LIN {X 0.189,Y -441.248,Z 653.481,A 0.000,B 0.000,C 90.000,E1 266.560} C_DIS
LIN {X -0.054,Y -433.305,Z 653.480,A 0.000,B 0.000,C 90.000,E1 266.388} C_DIS
LIN {X 0.144,Y -424.174,Z 653.479,A 0.000,B 0.000,C 90.000,E1 266.216} C_DIS
LIN {X 0.128,Y -416.575,Z 653.479,A 0.000,B 0.000,C 90.000,E1 266.159} C_DIS
LIN {X 0.071,Y -413.712,Z 653.479,A 0.000,B 0.000,C 90.000,E1 266.159} C_DIS
LIN {X 0.007,Y -180.928,Z 653.479,A 0.000,B 0.000,C 90.000,E1 266.159} C_DIS
LIN {X -0.082,Y -180.902,Z 653.474,A 0.000,B 0.000,C 90.000,E1 265.298} C_DIS
LIN {X 0.047,Y -180.232,Z 653.464,A 0.000,B 0.000,C 90.000,E1 263.571} C_DIS
LIN {X 0.064,Y -178.714,Z 653.441,A 0.000,B 0.000,C 90.000,E1 259.342} C_DIS
LIN {X -0.044,Y -175.764,Z 653.413,A 0.000,B 0.000,C 90.000,E1 254.283} C_DIS
LIN {X 0.006,Y -171.947,Z 653.384,A 0.000,B 0.000,C 90.000,E1 249.135} C_DIS
LIN {X -0.018,Y -171.334,Z 653.379,A 0.000,B 0.000,C 90.000,E1 248.284} C_DIS
LIN {X 0.034,Y -167.588,Z 653.355,A 0.000,B 0.000,C 90.000,E1 243.948} C_DIS
LIN {X -0.026,Y -166.226,Z 653.346,A 0.000,B 0.000,C 90.000,E1 242.231} C_DIS
LIN {X -0.038,Y -162.987,Z 653.326,A 0.000,B 0.000,C 90.000,E1 238.742} C_DIS
LIN {X 0.009,Y -160.904,Z 653.312,A 0.000,B 0.000,C 90.000,E1 236.087} C_DIS
LIN {X -0.013,Y -157.670,Z 653.292,A 0.000,B 0.000,C 90.000,E1 232.557} C_DIS
LIN {X -0.075,Y -155.708,Z 653.277,A 0.000,B 0.000,C 90.000,E1 229.908} C_DIS
LIN {X -0.020,Y -151.971,Z 653.252,A 0.000,B 0.000,C 90.000,E1 225.405} C_DIS
LIN {X -0.004,Y -150.213,Z 653.237,A 0.000,B 0.000,C 90.000,E1 222.690} C_DIS
LIN {X -0.079,Y -146.978,Z 653.212,A 0.000,B 0.000,C 90.000,E1 218.177} C_DIS
LIN {X 0.030,Y -145.565,Z 653.197,A 0.000,B 0.000,C 90.000,E1 215.391} C_DIS
LIN {X 0.029,Y -142.956,Z 653.171,A 0.000,B 0.000,C 90.000,E1 210.797} C_DIS
LIN {X -0.041,Y -141.582,Z 653.151,A 0.000,B 0.000,C 90.000,E1 207.129} C_DIS
LIN {X 0.007,Y -139.416,Z 653.115,A 0.000,B 0.000,C 90.000,E1 200.610} C_DIS
LIN {X 0.059,Y -139.142,Z 653.104,A 0.000,B 0.000,C 90.000,E1 198.725} C_DIS
LIN {X -0.050,Y -138.348,Z 653.057,A 0.000,B 0.000,C 90.000,E1 190.366} C_DIS
LIN {X -0.065,Y -139.491,Z 653.006,A 0.000,B 0.000,C 90.000,E1 181.031} C_DIS
LIN {X 0.015,Y -141.101,Z 652.975,A 0.000,B 0.000,C 90.000,E1 175.412} C_DIS
LIN {X -0.031,Y -142.479,Z 652.959,A 0.000,B 0.000,C 90.000,E1 172.648} C_DIS
LIN {X 0.058,Y -144.728,Z 652.933,A 0.000,B 0.000,C 90.000,E1 167.993} C_DIS
LIN {X 0.009,Y -147.332,Z 652.913,A 0.000,B 0.000,C 90.000,E1 164.338} C_DIS
LIN {X 0.074,Y -150.655,Z 652.888,A 0.000,B 0.000,C 90.000,E1 159.752} C_DIS
LIN {X -0.045,Y -154.133,Z 652.868,A 0.000,B 0.000,C 90.000,E1 156.177} C_DIS
LIN {X 0.018,Y -157.560,Z 652.848,A 0.000,B 0.000,C 90.000,E1 152.564} C_DIS
LIN {X 0.042,Y -161.803,Z 652.828,A 0.000,B 0.000,C 90.000,E1 148.997} C_DIS
LIN {X 0.062,Y -165.995,Z 652.808,A 0.000,B 0.000,C 90.000,E1 145.468} C_DIS
LIN {X 0.055,Y -170.992,Z 652.789,A 0.000,B 0.000,C 90.000,E1 141.984} C_DIS
LIN {X -0.029,Y -175.862,Z 652.770,A 0.000,B 0.000,C 90.000,E1 138.566} C_DIS
LIN {X -0.035,Y -181.467,Z 652.751,A 0.000,B 0.000,C 90.000,E1 135.162} C_DIS
LIN {X 0.101,Y -186.979,Z 652.732,A 0.000,B 0.000,C 90.000,E1 131.757} C_DIS
LIN {X -0.120,Y -191.043,Z 652.720,A 0.000,B 0.000,C 90.000,E1 129.644} C_DIS
LIN {X 0.173,Y -288.470,Z 652.720,A 0.000,B 0.000,C 90.000,E1 129.564} C_DIS
LIN {X 0.015,Y -290.425,Z 652.720,A 0.000,B 0.000,C 90.000,E1 129.564} C_DIS
LIN {X 0.087,Y -295.635,Z 652.718,A 0.000,B 0.000,C 90.000,E1 129.277} C_DIS
LIN {X -0.103,Y -298.817,Z 652.716,A 0.000,B 0.000,C 90.000,E1 128.991} C_DIS
LIN {X 0.074,Y -302.429,Z 652.713,A 0.000,B 0.000,C 90.000,E1 128.382} C_DIS
LIN {X -0.165,Y -303.887,Z 652.711,A 0.000,B 0.000,C 90.000,E1 128.096} C_DIS
LIN {X 0.022,Y -305.034,Z 652.710,A 0.000,B 0.000,C 90.000,E1 127.729} C_DIS
LIN {X 0.132,Y -315.593,Z 652.690,A 0.000,B 0.000,C 90.000,E1 124.119} C_DIS
LIN {X 0.009,Y -325.562,Z 652.674,A 0.000,B 0.000,C 90.000,E1 121.258} C_DIS
LIN {X -0.046,Y -336.851,Z 652.658,A 0.000,B 0.000,C 90.000,E1 118.437} C_DIS
LIN {X -0.093,Y -349.566,Z 652.643,A 0.000,B 0.000,C 90.000,E1 115.668} C_DIS
LIN {X -0.148,Y -362.154,Z 652.629,A 0.000,B 0.000,C 90.000,E1 113.259} C_DIS
LIN {X 0.024,Y -376.047,Z 652.616,A 0.000,B 0.000,C 90.000,E1 110.865} C_DIS
LIN {X 0.075,Y -391.345,Z 652.603,A 0.000,B 0.000,C 90.000,E1 108.544} C_DIS
LIN {X -0.132,Y -408.159,Z 652.591,A 0.000,B 0.000,C 90.000,E1 106.315} C_DIS
LIN {X -0.168,Y -426.613,Z 652.578,A 0.000,B 0.000,C 90.000,E1 104.120} C_DIS
LIN {X -0.103,Y -446.484,Z 652.567,A 0.000,B 0.000,C 90.000,E1 102.007} C_DIS
LIN {X -0.102,Y -466.963,Z 652.556,A 0.000,B 0.000,C 90.000,E1 100.074} C_DIS
LIN {X -0.128,Y -469.546,Z 652.555,A 0.000,B 0.000,C 90.000,E1 99.849} C_DIS
LIN {X -0.072,Y -471.802,Z 652.553,A 0.000,B 0.000,C 90.000,E1 99.613} C_DIS
LIN {X -0.186,Y -473.637,Z 652.552,A 0.000,B 0.000,C 90.000,E1 99.378} C_DIS
LIN {X 0.092,Y -475.022,Z 652.551,A 0.000,B 0.000,C 90.000,E1 99.095} C_DIS
LIN {X -0.185,Y -476.807,Z 652.548,A 0.000,B 0.000,C 90.000,E1 98.624} C_DIS
LIN {X -0.055,Y -477.505,Z 652.545,A 0.000,B 0.000,C 90.000,E1 98.106} C_DIS
LIN {X 0.087,Y -477.233,Z 652.542,A 0.000,B 0.000,C 90.000,E1 97.587} C_DIS
LIN {X -0.237,Y -475.951,Z 652.539,A 0.000,B 0.000,C 90.000,E1 97.125} C_DIS
LIN {X 0.100,Y -474.870,Z 652.538,A 0.000,B 0.000,C 90.000,E1 96.834} C_DIS
LIN {X -0.091,Y -473.421,Z 652.537,A 0.000,B 0.000,C 90.000,E1 96.606} C_DIS
LIN {X -0.133,Y -456.317,Z 652.523,A 0.000,B 0.000,C 90.000,E1 94.073} C_DIS
LIN {X 0.065,Y -445.602,Z 652.512,A 0.000,B 0.000,C 90.000,E1 92.236} C_DIS
LIN {X 0.026,Y -435.545,Z 652.502,A 0.000,B 0.000,C 90.000,E1 90.401} C_DIS
LIN {X 0.069,Y -426.626,Z 652.493,A 0.000,B 0.000,C 90.000,E1 88.797} C_DIS
LIN {X 0.061,Y -415.774,Z 652.483,A 0.000,B 0.000,C 90.000,E1 86.906} C_DIS
LIN {X 0.035,Y -401.764,Z 652.469,A 0.000,B 0.000,C 90.000,E1 84.432} C_DIS
LIN {X 0.082,Y -388.231,Z 652.455,A 0.000,B 0.000,C 90.000,E1 81.894} C_DIS
LIN {X -0.121,Y -375.167,Z 652.441,A 0.000,B 0.000,C 90.000,E1 79.342} C_DIS
LIN {X -0.091,Y -362.604,Z 652.426,A 0.000,B 0.000,C 90.000,E1 76.700} C_DIS
LIN {X 0.082,Y -348.061,Z 652.408,A 0.000,B 0.000,C 90.000,E1 73.378} C_DIS
LIN {X 0.057,Y -334.377,Z 652.389,A 0.000,B 0.000,C 90.000,E1 70.007} C_DIS
LIN {X 0.031,Y -321.830,Z 652.370,A 0.000,B 0.000,C 90.000,E1 66.561} C_DIS
LIN {X -0.103,Y -309.547,Z 652.348,A 0.000,B 0.000,C 90.000,E1 62.743} C_DIS
LIN {X 0.008,Y -300.306,Z 652.330,A 0.000,B 0.000,C 90.000,E1 59.459} C_DIS
LIN {X 0.042,Y -291.828,Z 652.312,A 0.000,B 0.000,C 90.000,E1 56.135} C_DIS
LIN {X 0.058,Y -283.710,Z 652.293,A 0.000,B 0.000,C 90.000,E1 52.763} C_DIS
LIN {X 0.008,Y -280.513,Z 652.286,A 0.000,B 0.000,C 90.000,E1 51.412} C_DIS
LIN {X -0.126,Y -277.134,Z 652.278,A 0.000,B 0.000,C 90.000,E1 50.070} C_DIS
LIN {X -0.128,Y -271.683,Z 652.267,A 0.000,B 0.000,C 90.000,E1 48.000} C_DIS
LIN {X -0.050,Y -265.784,Z 652.255,A 0.000,B 0.000,C 90.000,E1 45.891} C_DIS
LIN {X -0.089,Y -259.504,Z 652.243,A 0.000,B 0.000,C 90.000,E1 43.785} C_DIS
LIN {X 0.121,Y -252.929,Z 652.231,A 0.000,B 0.000,C 90.000,E1 41.595} C_DIS
LIN {X -0.104,Y -242.144,Z 652.211,A 0.000,B 0.000,C 90.000,E1 38.016} C_DIS
LIN {X 0.018,Y -234.162,Z 652.195,A 0.000,B 0.000,C 90.000,E1 35.025} C_DIS
LIN {X 0.056,Y -226.880,Z 652.178,A 0.000,B 0.000,C 90.000,E1 32.005} C_DIS
LIN {X 0.061,Y -220.310,Z 652.161,A 0.000,B 0.000,C 90.000,E1 28.949} C_DIS
LIN {X 0.078,Y -214.588,Z 652.144,A 0.000,B 0.000,C 90.000,E1 25.848} C_DIS
LIN {X 0.065,Y -209.634,Z 652.126,A 0.000,B 0.000,C 90.000,E1 22.717} C_DIS
LIN {X -0.026,Y -204.484,Z 652.104,A 0.000,B 0.000,C 90.000,E1 18.779} C_DIS
LIN {X -0.022,Y -200.459,Z 652.082,A 0.000,B 0.000,C 90.000,E1 14.773} C_DIS
LIN {X 0.038,Y -196.988,Z 652.055,A 0.000,B 0.000,C 90.000,E1 9.905} C_DIS
LIN {X 0.013,Y -194.464,Z 652.014,A 0.000,B 0.000,C 90.000,E1 2.579} C_DIS
LIN {X 0.002,Y -196.193,Z 651.961,A 0.000,B 0.000,C 90.000,E1 352.996} C_DIS
LIN {X 0.002,Y -199.224,Z 651.934,A 0.000,B 0.000,C 90.000,E1 348.117} C_DIS
LIN {X -0.079,Y -202.794,Z 651.912,A 0.000,B 0.000,C 90.000,E1 344.102} C_DIS
LIN {X 0.049,Y -207.381,Z 651.889,A 0.000,B 0.000,C 90.000,E1 340.061} C_DIS
LIN {X 0.033,Y -212.821,Z 651.867,A 0.000,B 0.000,C 90.000,E1 336.102} C_DIS
LIN {X -0.141,Y -218.987,Z 651.846,A 0.000,B 0.000,C 90.000,E1 332.231} C_DIS
LIN {X 0.089,Y -224.463,Z 651.828,A 0.000,B 0.000,C 90.000,E1 329.076} C_DIS
LIN {X 0.069,Y -231.711,Z 651.807,A 0.000,B 0.000,C 90.000,E1 325.261} C_DIS
LIN {X -0.086,Y -239.559,Z 651.786,A 0.000,B 0.000,C 90.000,E1 321.537} C_DIS
LIN {X 0.084,Y -248.181,Z 651.766,A 0.000,B 0.000,C 90.000,E1 317.796} C_DIS
LIN {X -0.049,Y -257.802,Z 651.745,A 0.000,B 0.000,C 90.000,E1 314.190} C_DIS
LIN {X -0.075,Y -267.404,Z 651.728,A 0.000,B 0.000,C 90.000,E1 310.987} C_DIS
LIN {X 0.177,Y -279.671,Z 651.708,A 0.000,B 0.000,C 90.000,E1 307.443} C_DIS
LIN {X -0.010,Y -293.237,Z 651.689,A 0.000,B 0.000,C 90.000,E1 304.072} C_DIS
LIN {X -0.002,Y -308.477,Z 651.671,A 0.000,B 0.000,C 90.000,E1 300.747} C_DIS
LIN {X -0.066,Y -323.517,Z 651.655,A 0.000,B 0.000,C 90.000,E1 297.847} C_DIS
LIN {X -0.144,Y -337.384,Z 651.641,A 0.000,B 0.000,C 90.000,E1 295.335} C_DIS
LIN {X 0.208,Y -355.656,Z 651.624,A 0.000,B 0.000,C 90.000,E1 292.206} C_DIS
LIN {X 0.158,Y -369.246,Z 651.612,A 0.000,B 0.000,C 90.000,E1 290.120} C_DIS
LIN {X -0.089,Y -384.236,Z 651.601,A 0.000,B 0.000,C 90.000,E1 288.109} C_DIS
LIN {X -0.200,Y -402.821,Z 651.588,A 0.000,B 0.000,C 90.000,E1 285.843} C_DIS
LIN {X -0.025,Y -414.425,Z 651.580,A 0.000,B 0.000,C 90.000,E1 284.426} C_DIS
LIN {X 0.081,Y -427.691,Z 651.571,A 0.000,B 0.000,C 90.000,E1 282.771} C_DIS
LIN {X 0.130,Y -438.189,Z 651.564,A 0.000,B 0.000,C 90.000,E1 281.422} C_DIS
LIN {X 0.108,Y -446.197,Z 651.558,A 0.000,B 0.000,C 90.000,E1 280.366} C_DIS
LIN {X 0.094,Y -454.150,Z 651.552,A 0.000,B 0.000,C 90.000,E1 279.321} C_DIS
LIN {X 0.057,Y -464.847,Z 651.545,A 0.000,B 0.000,C 90.000,E1 278.049} C_DIS
LIN {X -0.050,Y -470.598,Z 651.541,A 0.000,B 0.000,C 90.000,E1 277.296} C_DIS
LIN {X -0.104,Y -475.386,Z 651.536,A 0.000,B 0.000,C 90.000,E1 276.543} C_DIS
LIN {X -0.176,Y -479.394,Z 651.532,A 0.000,B 0.000,C 90.000,E1 275.796} C_DIS
LIN {X -0.027,Y -481.609,Z 651.529,A 0.000,B 0.000,C 90.000,E1 275.277} C_DIS
LIN {X 0.138,Y -483.468,Z 651.527,A 0.000,B 0.000,C 90.000,E1 274.759} C_DIS
LIN {X -0.213,Y -484.886,Z 651.524,A 0.000,B 0.000,C 90.000,E1 274.302} C_DIS
LIN {X -0.033,Y -485.902,Z 651.521,A 0.000,B 0.000,C 90.000,E1 273.784} C_DIS
LIN {X 0.125,Y -486.560,Z 651.518,A 0.000,B 0.000,C 90.000,E1 273.269} C_DIS
LIN {X -0.169,Y -486.874,Z 651.516,A 0.000,B 0.000,C 90.000,E1 272.808} C_DIS
LIN {X 0.002,Y -486.931,Z 651.513,A 0.000,B 0.000,C 90.000,E1 272.293} C_DIS
LIN {X 0.193,Y -486.719,Z 651.510,A 0.000,B 0.000,C 90.000,E1 271.776} C_DIS
LIN {X -0.120,Y -486.113,Z 651.507,A 0.000,B 0.000,C 90.000,E1 271.318} C_DIS
LIN {X 0.055,Y -485.118,Z 651.505,A 0.000,B 0.000,C 90.000,E1 270.802} C_DIS
LIN {X 0.226,Y -483.673,Z 651.502,A 0.000,B 0.000,C 90.000,E1 270.286} C_DIS
LIN {X -0.091,Y -481.651,Z 651.499,A 0.000,B 0.000,C 90.000,E1 269.828} C_DIS
LIN {X 0.066,Y -478.997,Z 651.496,A 0.000,B 0.000,C 90.000,E1 269.312} C_DIS
LIN {X 0.201,Y -475.487,Z 651.493,A 0.000,B 0.000,C 90.000,E1 268.797} C_DIS
LIN {X -0.156,Y -471.011,Z 651.491,A 0.000,B 0.000,C 90.000,E1 268.339} C_DIS
LIN {X 0.140,Y -468.359,Z 651.489,A 0.000,B 0.000,C 90.000,E1 268.051} C_DIS
LIN {X 0.024,Y -462.383,Z 651.487,A 0.000,B 0.000,C 90.000,E1 267.593} C_DIS
LIN {X 0.093,Y -459.096,Z 651.485,A 0.000,B 0.000,C 90.000,E1 267.364} C_DIS
LIN {X -0.043,Y -455.866,Z 651.484,A 0.000,B 0.000,C 90.000,E1 267.192} C_DIS
LIN {X 0.011,Y -448.763,Z 651.482,A 0.000,B 0.000,C 90.000,E1 266.846} C_DIS
LIN {X 0.165,Y -441.242,Z 651.481,A 0.000,B 0.000,C 90.000,E1 266.560} C_DIS
LIN {X -0.067,Y -433.363,Z 651.480,A 0.000,B 0.000,C 90.000,E1 266.388} C_DIS
LIN {X 0.125,Y -423.997,Z 651.479,A 0.000,B 0.000,C 90.000,E1 266.216} C_DIS
LIN {X 0.109,Y -415.978,Z 651.479,A 0.000,B 0.000,C 90.000,E1 266.159} C_DIS
LIN {X 0.052,Y -412.268,Z 651.479,A 0.000,B 0.000,C 90.000,E1 266.159} C_DIS
LIN {X -0.001,Y -180.927,Z 651.479,A 0.000,B 0.000,C 90.000,E1 266.159} C_DIS
LIN {X -0.088,Y -180.902,Z 651.474,A 0.000,B 0.000,C 90.000,E1 265.298} C_DIS
LIN {X 0.041,Y -180.231,Z 651.464,A 0.000,B 0.000,C 90.000,E1 263.571} C_DIS
LIN {X 0.058,Y -178.714,Z 651.441,A 0.000,B 0.000,C 90.000,E1 259.342} C_DIS
LIN {X -0.051,Y -175.762,Z 651.413,A 0.000,B 0.000,C 90.000,E1 254.283} C_DIS
LIN {X -0.001,Y -171.946,Z 651.384,A 0.000,B 0.000,C 90.000,E1 249.135} C_DIS
LIN {X -0.024,Y -171.332,Z 651.379,A 0.000,B 0.000,C 90.000,E1 248.284} C_DIS
LIN {X 0.029,Y -167.586,Z 651.355,A 0.000,B 0.000,C 90.000,E1 243.948} C_DIS
LIN {X -0.032,Y -166.224,Z 651.346,A 0.000,B 0.000,C 90.000,E1 242.231} C_DIS
LIN {X -0.044,Y -162.986,Z 651.326,A 0.000,B 0.000,C 90.000,E1 238.742} C_DIS
LIN {X 0.003,Y -160.901,Z 651.312,A 0.000,B 0.000,C 90.000,E1 236.087} C_DIS
LIN {X -0.018,Y -157.668,Z 651.292,A 0.000,B 0.000,C 90.000,E1 232.557} C_DIS
LIN {X -0.080,Y -155.706,Z 651.277,A 0.000,B 0.000,C 90.000,E1 229.908} C_DIS
LIN {X -0.026,Y -151.969,Z 651.252,A 0.000,B 0.000,C 90.000,E1 225.405} C_DIS
LIN {X -0.009,Y -150.211,Z 651.237,A 0.000,B 0.000,C 90.000,E1 222.690} C_DIS
LIN {X -0.085,Y -146.977,Z 651.212,A 0.000,B 0.000,C 90.000,E1 218.177} C_DIS
LIN {X 0.024,Y -145.563,Z 651.197,A 0.000,B 0.000,C 90.000,E1 215.391} C_DIS
LIN {X 0.023,Y -142.955,Z 651.171,A 0.000,B 0.000,C 90.000,E1 210.797} C_DIS
LIN {X -0.046,Y -141.581,Z 651.151,A 0.000,B 0.000,C 90.000,E1 207.129} C_DIS
LIN {X 0.002,Y -139.416,Z 651.115,A 0.000,B 0.000,C 90.000,E1 200.610} C_DIS
LIN {X 0.053,Y -139.141,Z 651.104,A 0.000,B 0.000,C 90.000,E1 198.725} C_DIS
LIN {X -0.055,Y -138.348,Z 651.057,A 0.000,B 0.000,C 90.000,E1 190.366} C_DIS
LIN {X 0.069,Y -139.491,Z 651.006,A 0.000,B 0.000,C 90.000,E1 180.974} C_DIS
LIN {X 0.010,Y -141.102,Z 650.975,A 0.000,B 0.000,C 90.000,E1 175.412} C_DIS
LIN {X -0.037,Y -142.480,Z 650.959,A 0.000,B 0.000,C 90.000,E1 172.648} C_DIS
LIN {X 0.052,Y -144.729,Z 650.933,A 0.000,B 0.000,C 90.000,E1 167.993} C_DIS
LIN {X 0.003,Y -147.334,Z 650.913,A 0.000,B 0.000,C 90.000,E1 164.338} C_DIS
LIN {X 0.068,Y -150.656,Z 650.888,A 0.000,B 0.000,C 90.000,E1 159.752} C_DIS
LIN {X -0.051,Y -154.135,Z 650.868,A 0.000,B 0.000,C 90.000,E1 156.177} C_DIS
LIN {X 0.012,Y -157.563,Z 650.848,A 0.000,B 0.000,C 90.000,E1 152.564} C_DIS
LIN {X 0.037,Y -161.806,Z 650.828,A 0.000,B 0.000,C 90.000,E1 148.997} C_DIS
LIN {X 0.056,Y -165.998,Z 650.808,A 0.000,B 0.000,C 90.000,E1 145.468} C_DIS
LIN {X 0.048,Y -170.995,Z 650.789,A 0.000,B 0.000,C 90.000,E1 141.984} C_DIS
LIN {X -0.036,Y -175.865,Z 650.770,A 0.000,B 0.000,C 90.000,E1 138.566} C_DIS
LIN {X -0.042,Y -181.470,Z 650.751,A 0.000,B 0.000,C 90.000,E1 135.162} C_DIS
LIN {X 0.094,Y -186.982,Z 650.732,A 0.000,B 0.000,C 90.000,E1 131.757} C_DIS
LIN {X -0.127,Y -191.046,Z 650.720,A 0.000,B 0.000,C 90.000,E1 129.644} C_DIS
LIN {X 0.162,Y -288.697,Z 650.720,A 0.000,B 0.000,C 90.000,E1 129.564} C_DIS
LIN {X 0.005,Y -290.478,Z 650.720,A 0.000,B 0.000,C 90.000,E1 129.564} C_DIS
LIN {X 0.077,Y -295.638,Z 650.718,A 0.000,B 0.000,C 90.000,E1 129.277} C_DIS
LIN {X 0.059,Y -298.836,Z 650.716,A 0.000,B 0.000,C 90.000,E1 128.955} C_DIS
LIN {X 0.038,Y -302.443,Z 650.713,A 0.000,B 0.000,C 90.000,E1 128.382} C_DIS
LIN {X 0.039,Y -303.894,Z 650.711,A 0.000,B 0.000,C 90.000,E1 128.051} C_DIS
LIN {X -0.014,Y -305.035,Z 650.710,A 0.000,B 0.000,C 90.000,E1 127.729} C_DIS
LIN {X 0.095,Y -315.593,Z 650.690,A 0.000,B 0.000,C 90.000,E1 124.119} C_DIS
LIN {X -0.029,Y -325.566,Z 650.674,A 0.000,B 0.000,C 90.000,E1 121.258} C_DIS
LIN {X -0.085,Y -336.857,Z 650.658,A 0.000,B 0.000,C 90.000,E1 118.437} C_DIS
LIN {X -0.134,Y -349.576,Z 650.642,A 0.000,B 0.000,C 90.000,E1 115.668} C_DIS
LIN {X 0.142,Y -362.168,Z 650.629,A 0.000,B 0.000,C 90.000,E1 113.206} C_DIS
LIN {X -0.019,Y -376.064,Z 650.616,A 0.000,B 0.000,C 90.000,E1 110.865} C_DIS
LIN {X 0.030,Y -391.366,Z 650.603,A 0.000,B 0.000,C 90.000,E1 108.544} C_DIS
LIN {X -0.178,Y -408.183,Z 650.591,A 0.000,B 0.000,C 90.000,E1 106.315} C_DIS
LIN {X 0.198,Y -426.642,Z 650.578,A 0.000,B 0.000,C 90.000,E1 104.064} C_DIS
LIN {X -0.150,Y -446.516,Z 650.567,A 0.000,B 0.000,C 90.000,E1 102.007} C_DIS
LIN {X -0.149,Y -466.996,Z 650.556,A 0.000,B 0.000,C 90.000,E1 100.074} C_DIS
LIN {X -0.174,Y -469.579,Z 650.555,A 0.000,B 0.000,C 90.000,E1 99.849} C_DIS
LIN {X -0.118,Y -471.851,Z 650.553,A 0.000,B 0.000,C 90.000,E1 99.613} C_DIS
LIN {X 0.243,Y -473.691,Z 650.552,A 0.000,B 0.000,C 90.000,E1 99.321} C_DIS
LIN {X 0.062,Y -475.080,Z 650.551,A 0.000,B 0.000,C 90.000,E1 99.095} C_DIS
LIN {X -0.215,Y -476.883,Z 650.548,A 0.000,B 0.000,C 90.000,E1 98.624} C_DIS
LIN {X -0.084,Y -477.595,Z 650.545,A 0.000,B 0.000,C 90.000,E1 98.106} C_DIS
LIN {X 0.059,Y -477.335,Z 650.542,A 0.000,B 0.000,C 90.000,E1 97.587} C_DIS
LIN {X 0.207,Y -476.068,Z 650.539,A 0.000,B 0.000,C 90.000,E1 97.068} C_DIS
LIN {X 0.072,Y -474.996,Z 650.538,A 0.000,B 0.000,C 90.000,E1 96.834} C_DIS
LIN {X -0.118,Y -473.559,Z 650.537,A 0.000,B 0.000,C 90.000,E1 96.606} C_DIS
LIN {X -0.156,Y -456.421,Z 650.523,A 0.000,B 0.000,C 90.000,E1 94.073} C_DIS
LIN {X -0.153,Y -447.148,Z 650.514,A 0.000,B 0.000,C 90.000,E1 92.522} C_DIS
LIN {X 0.008,Y -435.627,Z 650.502,A 0.000,B 0.000,C 90.000,E1 90.401} C_DIS
LIN {X 0.052,Y -426.729,Z 650.493,A 0.000,B 0.000,C 90.000,E1 88.797} C_DIS
LIN {X 0.046,Y -415.859,Z 650.483,A 0.000,B 0.000,C 90.000,E1 86.906} C_DIS
LIN {X -0.068,Y -403.383,Z 650.471,A 0.000,B 0.000,C 90.000,E1 84.723} C_DIS
LIN {X 0.022,Y -389.812,Z 650.457,A 0.000,B 0.000,C 90.000,E1 82.186} C_DIS
LIN {X -0.145,Y -376.703,Z 650.442,A 0.000,B 0.000,C 90.000,E1 79.634} C_DIS
LIN {X -0.055,Y -365.478,Z 650.429,A 0.000,B 0.000,C 90.000,E1 77.285} C_DIS
LIN {X 0.091,Y -352.055,Z 650.413,A 0.000,B 0.000,C 90.000,E1 74.283} C_DIS
LIN {X -0.130,Y -340.624,Z 650.398,A 0.000,B 0.000,C 90.000,E1 71.583} C_DIS
LIN {X -0.089,Y -326.441,Z 650.377,A 0.000,B 0.000,C 90.000,E1 67.847} C_DIS
LIN {X -0.041,Y -313.677,Z 650.356,A 0.000,B 0.000,C 90.000,E1 64.024} C_DIS
LIN {X -0.097,Y -304.115,Z 650.338,A 0.000,B 0.000,C 90.000,E1 60.795} C_DIS
LIN {X 0.143,Y -295.365,Z 650.319,A 0.000,B 0.000,C 90.000,E1 57.454} C_DIS
LIN {X -0.035,Y -288.728,Z 650.305,A 0.000,B 0.000,C 90.000,E1 54.815} C_DIS
LIN {X -0.036,Y -282.321,Z 650.289,A 0.000,B 0.000,C 90.000,E1 52.110} C_DIS
LIN {X -0.086,Y -277.345,Z 650.278,A 0.000,B 0.000,C 90.000,E1 50.070} C_DIS
LIN {X -0.086,Y -271.918,Z 650.267,A 0.000,B 0.000,C 90.000,E1 48.000} C_DIS
LIN {X -0.003,Y -266.013,Z 650.255,A 0.000,B 0.000,C 90.000,E1 45.891} C_DIS
LIN {X -0.040,Y -259.713,Z 650.243,A 0.000,B 0.000,C 90.000,E1 43.785} C_DIS
LIN {X 0.005,Y -253.128,Z 650.231,A 0.000,B 0.000,C 90.000,E1 41.634} C_DIS
LIN {X -0.068,Y -242.310,Z 650.211,A 0.000,B 0.000,C 90.000,E1 38.016} C_DIS
LIN {X 0.057,Y -234.316,Z 650.195,A 0.000,B 0.000,C 90.000,E1 35.025} C_DIS
LIN {X 0.098,Y -227.040,Z 650.178,A 0.000,B 0.000,C 90.000,E1 32.005} C_DIS
LIN {X 0.105,Y -220.458,Z 650.161,A 0.000,B 0.000,C 90.000,E1 28.949} C_DIS
LIN {X -0.069,Y -214.745,Z 650.144,A 0.000,B 0.000,C 90.000,E1 25.899} C_DIS
LIN {X -0.079,Y -209.772,Z 650.126,A 0.000,B 0.000,C 90.000,E1 22.770} C_DIS
LIN {X 0.026,Y -204.611,Z 650.104,A 0.000,B 0.000,C 90.000,E1 18.779} C_DIS
LIN {X 0.032,Y -200.568,Z 650.082,A 0.000,B 0.000,C 90.000,E1 14.773} C_DIS
LIN {X 0.097,Y -197.096,Z 650.055,A 0.000,B 0.000,C 90.000,E1 9.905} C_DIS
LIN {X 0.076,Y -194.560,Z 650.014,A 0.000,B 0.000,C 90.000,E1 2.579} C_DIS
LIN {X 0.007,Y -196.283,Z 649.961,A 0.000,B 0.000,C 90.000,E1 352.996} C_DIS
LIN {X 0.010,Y -199.297,Z 649.934,A 0.000,B 0.000,C 90.000,E1 348.117} C_DIS
LIN {X -0.069,Y -202.859,Z 649.912,A 0.000,B 0.000,C 90.000,E1 344.102} C_DIS
LIN {X 0.061,Y -207.438,Z 649.889,A 0.000,B 0.000,C 90.000,E1 340.061} C_DIS
LIN {X 0.048,Y -212.879,Z 649.867,A 0.000,B 0.000,C 90.000,E1 336.102} C_DIS
LIN {X -0.123,Y -219.042,Z 649.846,A 0.000,B 0.000,C 90.000,E1 332.231} C_DIS
LIN {X 0.024,Y -225.908,Z 649.824,A 0.000,B 0.000,C 90.000,E1 328.329} C_DIS
LIN {X -0.010,Y -233.263,Z 649.803,A 0.000,B 0.000,C 90.000,E1 324.529} C_DIS
LIN {X -0.113,Y -241.219,Z 649.782,A 0.000,B 0.000,C 90.000,E1 320.803} C_DIS
LIN {X 0.091,Y -250.009,Z 649.762,A 0.000,B 0.000,C 90.000,E1 317.067} C_DIS
LIN {X 0.019,Y -259.796,Z 649.741,A 0.000,B 0.000,C 90.000,E1 313.461} C_DIS
LIN {X 0.084,Y -269.691,Z 649.724,A 0.000,B 0.000,C 90.000,E1 310.253} C_DIS
LIN {X 0.027,Y -282.198,Z 649.704,A 0.000,B 0.000,C 90.000,E1 306.790} C_DIS
LIN {X 0.161,Y -294.625,Z 649.687,A 0.000,B 0.000,C 90.000,E1 303.706} C_DIS
LIN {X 0.055,Y -309.988,Z 649.669,A 0.000,B 0.000,C 90.000,E1 300.413} C_DIS
LIN {X 0.040,Y -325.137,Z 649.653,A 0.000,B 0.000,C 90.000,E1 297.513} C_DIS
LIN {X -0.144,Y -339.032,Z 649.639,A 0.000,B 0.000,C 90.000,E1 295.027} C_DIS
LIN {X -0.105,Y -355.568,Z 649.624,A 0.000,B 0.000,C 90.000,E1 292.259} C_DIS
LIN {X 0.173,Y -369.166,Z 649.612,A 0.000,B 0.000,C 90.000,E1 290.120} C_DIS
LIN {X -0.075,Y -384.158,Z 649.601,A 0.000,B 0.000,C 90.000,E1 288.109} C_DIS
LIN {X -0.188,Y -402.724,Z 649.588,A 0.000,B 0.000,C 90.000,E1 285.843} C_DIS
LIN {X -0.013,Y -414.332,Z 649.580,A 0.000,B 0.000,C 90.000,E1 284.426} C_DIS
LIN {X 0.091,Y -427.596,Z 649.571,A 0.000,B 0.000,C 90.000,E1 282.771} C_DIS
LIN {X 0.139,Y -438.116,Z 649.564,A 0.000,B 0.000,C 90.000,E1 281.422} C_DIS
LIN {X 0.115,Y -446.141,Z 649.558,A 0.000,B 0.000,C 90.000,E1 280.366} C_DIS
LIN {X 0.101,Y -454.094,Z 649.552,A 0.000,B 0.000,C 90.000,E1 279.321} C_DIS
LIN {X 0.182,Y -462.829,Z 649.546,A 0.000,B 0.000,C 90.000,E1 278.276} C_DIS
LIN {X 0.002,Y -468.788,Z 649.542,A 0.000,B 0.000,C 90.000,E1 277.530} C_DIS
LIN {X -0.070,Y -473.893,Z 649.538,A 0.000,B 0.000,C 90.000,E1 276.777} C_DIS
LIN {X -0.148,Y -478.142,Z 649.533,A 0.000,B 0.000,C 90.000,E1 276.030} C_DIS
LIN {X -0.144,Y -481.600,Z 649.529,A 0.000,B 0.000,C 90.000,E1 275.277} C_DIS
LIN {X 0.019,Y -483.443,Z 649.526,A 0.000,B 0.000,C 90.000,E1 274.759} C_DIS
LIN {X 0.151,Y -484.862,Z 649.524,A 0.000,B 0.000,C 90.000,E1 274.245} C_DIS
LIN {X -0.152,Y -485.869,Z 649.521,A 0.000,B 0.000,C 90.000,E1 273.784} C_DIS
LIN {X 0.005,Y -486.498,Z 649.518,A 0.000,B 0.000,C 90.000,E1 273.269} C_DIS
LIN {X 0.197,Y -486.830,Z 649.515,A 0.000,B 0.000,C 90.000,E1 272.751} C_DIS
LIN {X -0.119,Y -486.863,Z 649.513,A 0.000,B 0.000,C 90.000,E1 272.293} C_DIS
LIN {X 0.073,Y -486.602,Z 649.510,A 0.000,B 0.000,C 90.000,E1 271.776} C_DIS
LIN {X -0.240,Y -486.036,Z 649.507,A 0.000,B 0.000,C 90.000,E1 271.318} C_DIS
LIN {X -0.066,Y -485.046,Z 649.504,A 0.000,B 0.000,C 90.000,E1 270.802} C_DIS
LIN {X 0.105,Y -483.624,Z 649.502,A 0.000,B 0.000,C 90.000,E1 270.286} C_DIS
LIN {X -0.212,Y -481.597,Z 649.499,A 0.000,B 0.000,C 90.000,E1 269.828} C_DIS
LIN {X -0.056,Y -478.895,Z 649.496,A 0.000,B 0.000,C 90.000,E1 269.312} C_DIS
LIN {X 0.081,Y -475.370,Z 649.493,A 0.000,B 0.000,C 90.000,E1 268.797} C_DIS
LIN {X -0.098,Y -473.294,Z 649.492,A 0.000,B 0.000,C 90.000,E1 268.568} C_DIS
LIN {X 0.021,Y -468.206,Z 649.489,A 0.000,B 0.000,C 90.000,E1 268.051} C_DIS
LIN {X -0.166,Y -465.199,Z 649.488,A 0.000,B 0.000,C 90.000,E1 267.822} C_DIS
LIN {X -0.043,Y -458.862,Z 649.485,A 0.000,B 0.000,C 90.000,E1 267.364} C_DIS
LIN {X -0.163,Y -455.679,Z 649.484,A 0.000,B 0.000,C 90.000,E1 267.192} C_DIS
LIN {X -0.075,Y -448.576,Z 649.482,A 0.000,B 0.000,C 90.000,E1 266.846} C_DIS
LIN {X 0.096,Y -441.032,Z 649.481,A 0.000,B 0.000,C 90.000,E1 266.560} C_DIS
LIN {X -0.128,Y -433.074,Z 649.480,A 0.000,B 0.000,C 90.000,E1 266.388} C_DIS
LIN {X 0.087,Y -428.368,Z 649.479,A 0.000,B 0.000,C 90.000,E1 266.274} C_DIS
LIN {X -0.143,Y -419.904,Z 649.479,A 0.000,B 0.000,C 90.000,E1 266.216} C_DIS
LIN {X 0.060,Y -413.336,Z 649.479,A 0.000,B 0.000,C 90.000,E1 266.159} C_DIS
LIN {X 0.004,Y -180.927,Z 649.479,A 0.000,B 0.000,C 90.000,E1 266.159} C_DIS
LIN {X -0.089,Y -180.902,Z 649.474,A 0.000,B 0.000,C 90.000,E1 265.298} C_DIS
LIN {X 0.040,Y -180.231,Z 649.464,A 0.000,B 0.000,C 90.000,E1 263.571} C_DIS
LIN {X 0.057,Y -178.714,Z 649.441,A 0.000,B 0.000,C 90.000,E1 259.342} C_DIS
LIN {X -0.051,Y -175.762,Z 649.413,A 0.000,B 0.000,C 90.000,E1 254.283} C_DIS
LIN {X -0.001,Y -171.946,Z 649.384,A 0.000,B 0.000,C 90.000,E1 249.135} C_DIS
LIN {X -0.025,Y -171.332,Z 649.379,A 0.000,B 0.000,C 90.000,E1 248.284} C_DIS
LIN {X 0.028,Y -167.587,Z 649.355,A 0.000,B 0.000,C 90.000,E1 243.948} C_DIS
LIN {X -0.034,Y -166.223,Z 649.346,A 0.000,B 0.000,C 90.000,E1 242.231} C_DIS
LIN {X -0.045,Y -162.985,Z 649.326,A 0.000,B 0.000,C 90.000,E1 238.742} C_DIS
LIN {X 0.003,Y -160.901,Z 649.312,A 0.000,B 0.000,C 90.000,E1 236.087} C_DIS
LIN {X -0.020,Y -157.668,Z 649.292,A 0.000,B 0.000,C 90.000,E1 232.557} C_DIS
LIN {X -0.081,Y -155.707,Z 649.277,A 0.000,B 0.000,C 90.000,E1 229.908} C_DIS
LIN {X -0.026,Y -151.969,Z 649.252,A 0.000,B 0.000,C 90.000,E1 225.405} C_DIS
LIN {X -0.010,Y -150.210,Z 649.237,A 0.000,B 0.000,C 90.000,E1 222.690} C_DIS
LIN {X -0.086,Y -146.977,Z 649.212,A 0.000,B 0.000,C 90.000,E1 218.177} C_DIS
LIN {X 0.024,Y -145.563,Z 649.197,A 0.000,B 0.000,C 90.000,E1 215.391} C_DIS
LIN {X 0.023,Y -142.955,Z 649.171,A 0.000,B 0.000,C 90.000,E1 210.797} C_DIS
LIN {X -0.047,Y -141.581,Z 649.151,A 0.000,B 0.000,C 90.000,E1 207.129} C_DIS
LIN {X 0.001,Y -139.416,Z 649.115,A 0.000,B 0.000,C 90.000,E1 200.610} C_DIS
LIN {X 0.053,Y -139.141,Z 649.104,A 0.000,B 0.000,C 90.000,E1 198.725} C_DIS
LIN {X -0.056,Y -138.348,Z 649.057,A 0.000,B 0.000,C 90.000,E1 190.366} C_DIS
LIN {X 0.068,Y -139.491,Z 649.006,A 0.000,B 0.000,C 90.000,E1 180.974} C_DIS
LIN {X 0.009,Y -141.102,Z 648.975,A 0.000,B 0.000,C 90.000,E1 175.412} C_DIS
LIN {X -0.038,Y -142.480,Z 648.959,A 0.000,B 0.000,C 90.000,E1 172.648} C_DIS
LIN {X 0.052,Y -144.729,Z 648.933,A 0.000,B 0.000,C 90.000,E1 167.993} C_DIS
LIN {X 0.002,Y -147.334,Z 648.913,A 0.000,B 0.000,C 90.000,E1 164.338} C_DIS
LIN {X 0.067,Y -150.657,Z 648.888,A 0.000,B 0.000,C 90.000,E1 159.752} C_DIS
LIN {X -0.051,Y -154.135,Z 648.868,A 0.000,B 0.000,C 90.000,E1 156.177} C_DIS
LIN {X 0.011,Y -157.563,Z 648.848,A 0.000,B 0.000,C 90.000,E1 152.564} C_DIS
LIN {X 0.036,Y -161.806,Z 648.828,A 0.000,B 0.000,C 90.000,E1 148.997} C_DIS
LIN {X 0.055,Y -165.997,Z 648.808,A 0.000,B 0.000,C 90.000,E1 145.468} C_DIS
LIN {X 0.047,Y -170.996,Z 648.789,A 0.000,B 0.000,C 90.000,E1 141.984} C_DIS
LIN {X -0.036,Y -175.866,Z 648.770,A 0.000,B 0.000,C 90.000,E1 138.566} C_DIS
LIN {X -0.043,Y -181.470,Z 648.751,A 0.000,B 0.000,C 90.000,E1 135.162} C_DIS
LIN {X 0.094,Y -186.982,Z 648.732,A 0.000,B 0.000,C 90.000,E1 131.757} C_DIS
LIN {X -0.127,Y -191.046,Z 648.720,A 0.000,B 0.000,C 90.000,E1 129.644} C_DIS
LIN {X 0.162,Y -288.888,Z 648.720,A 0.000,B 0.000,C 90.000,E1 129.564} C_DIS
LIN {X 0.004,Y -290.532,Z 648.720,A 0.000,B 0.000,C 90.000,E1 129.564} C_DIS
LIN {X 0.077,Y -295.638,Z 648.718,A 0.000,B 0.000,C 90.000,E1 129.277} C_DIS
LIN {X 0.041,Y -298.852,Z 648.716,A 0.000,B 0.000,C 90.000,E1 128.955} C_DIS
LIN {X 0.010,Y -302.453,Z 648.713,A 0.000,B 0.000,C 90.000,E1 128.382} C_DIS
LIN {X 0.009,Y -303.897,Z 648.711,A 0.000,B 0.000,C 90.000,E1 128.051} C_DIS
LIN {X -0.043,Y -305.031,Z 648.710,A 0.000,B 0.000,C 90.000,E1 127.729} C_DIS
LIN {X 0.065,Y -315.591,Z 648.690,A 0.000,B 0.000,C 90.000,E1 124.119} C_DIS
LIN {X -0.061,Y -325.565,Z 648.674,A 0.000,B 0.000,C 90.000,E1 121.258} C_DIS
LIN {X 0.043,Y -336.859,Z 648.658,A 0.000,B 0.000,C 90.000,E1 118.409} C_DIS
LIN {X -0.017,Y -349.581,Z 648.642,A 0.000,B 0.000,C 90.000,E1 115.643} C_DIS
LIN {X 0.107,Y -362.175,Z 648.629,A 0.000,B 0.000,C 90.000,E1 113.206} C_DIS
LIN {X -0.055,Y -376.074,Z 648.616,A 0.000,B 0.000,C 90.000,E1 110.865} C_DIS
LIN {X -0.007,Y -391.378,Z 648.603,A 0.000,B 0.000,C 90.000,E1 108.544} C_DIS
LIN {X 0.175,Y -408.200,Z 648.590,A 0.000,B 0.000,C 90.000,E1 106.260} C_DIS
LIN {X 0.159,Y -426.661,Z 648.578,A 0.000,B 0.000,C 90.000,E1 104.064} C_DIS
LIN {X -0.190,Y -446.538,Z 648.567,A 0.000,B 0.000,C 90.000,E1 102.007} C_DIS
LIN {X -0.188,Y -467.020,Z 648.556,A 0.000,B 0.000,C 90.000,E1 100.074} C_DIS
LIN {X -0.156,Y -471.890,Z 648.553,A 0.000,B 0.000,C 90.000,E1 99.613} C_DIS
LIN {X 0.213,Y -473.737,Z 648.552,A 0.000,B 0.000,C 90.000,E1 99.321} C_DIS
LIN {X 0.041,Y -475.132,Z 648.551,A 0.000,B 0.000,C 90.000,E1 99.095} C_DIS
LIN {X 0.237,Y -476.954,Z 648.548,A 0.000,B 0.000,C 90.000,E1 98.568} C_DIS
LIN {X -0.105,Y -477.681,Z 648.545,A 0.000,B 0.000,C 90.000,E1 98.106} C_DIS
LIN {X 0.038,Y -477.436,Z 648.542,A 0.000,B 0.000,C 90.000,E1 97.587} C_DIS
LIN {X 0.187,Y -476.186,Z 648.539,A 0.000,B 0.000,C 90.000,E1 97.068} C_DIS
LIN {X 0.053,Y -475.124,Z 648.538,A 0.000,B 0.000,C 90.000,E1 96.834} C_DIS
LIN {X -0.137,Y -473.698,Z 648.537,A 0.000,B 0.000,C 90.000,E1 96.606} C_DIS
LIN {X -0.138,Y -456.522,Z 648.523,A 0.000,B 0.000,C 90.000,E1 94.069} C_DIS
LIN {X 0.032,Y -445.781,Z 648.512,A 0.000,B 0.000,C 90.000,E1 92.236} C_DIS
LIN {X 0.159,Y -434.272,Z 648.501,A 0.000,B 0.000,C 90.000,E1 90.115} C_DIS
LIN {X 0.044,Y -426.827,Z 648.493,A 0.000,B 0.000,C 90.000,E1 88.797} C_DIS
LIN {X -0.060,Y -417.521,Z 648.484,A 0.000,B 0.000,C 90.000,E1 87.192} C_DIS
LIN {X -0.127,Y -405.031,Z 648.472,A 0.000,B 0.000,C 90.000,E1 85.008} C_DIS
LIN {X 0.013,Y -391.395,Z 648.458,A 0.000,B 0.000,C 90.000,E1 82.470} C_DIS
LIN {X -0.162,Y -378.263,Z 648.444,A 0.000,B 0.000,C 90.000,E1 79.926} C_DIS
LIN {X -0.114,Y -366.997,Z 648.431,A 0.000,B 0.000,C 90.000,E1 77.589} C_DIS
LIN {X 0.212,Y -354.768,Z 648.416,A 0.000,B 0.000,C 90.000,E1 74.866} C_DIS
LIN {X -0.032,Y -343.279,Z 648.401,A 0.000,B 0.000,C 90.000,E1 72.181} C_DIS
LIN {X -0.012,Y -328.880,Z 648.380,A 0.000,B 0.000,C 90.000,E1 68.465} C_DIS
LIN {X -0.014,Y -315.906,Z 648.359,A 0.000,B 0.000,C 90.000,E1 64.665} C_DIS
LIN {X -0.004,Y -306.167,Z 648.341,A 0.000,B 0.000,C 90.000,E1 61.435} C_DIS
LIN {X 0.153,Y -297.251,Z 648.323,A 0.000,B 0.000,C 90.000,E1 58.122} C_DIS
LIN {X 0.004,Y -288.927,Z 648.305,A 0.000,B 0.000,C 90.000,E1 54.815} C_DIS
LIN {X 0.006,Y -282.513,Z 648.289,A 0.000,B 0.000,C 90.000,E1 52.110} C_DIS
LIN {X -0.041,Y -277.555,Z 648.278,A 0.000,B 0.000,C 90.000,E1 50.070} C_DIS
LIN {X -0.037,Y -272.143,Z 648.267,A 0.000,B 0.000,C 90.000,E1 48.000} C_DIS
LIN {X 0.048,Y -266.257,Z 648.255,A 0.000,B 0.000,C 90.000,E1 45.891} C_DIS
LIN {X 0.014,Y -259.931,Z 648.243,A 0.000,B 0.000,C 90.000,E1 43.785} C_DIS
LIN {X -0.127,Y -253.327,Z 648.231,A 0.000,B 0.000,C 90.000,E1 41.676} C_DIS
LIN {X -0.007,Y -242.478,Z 648.211,A 0.000,B 0.000,C 90.000,E1 38.016} C_DIS
LIN {X 0.120,Y -234.483,Z 648.195,A 0.000,B 0.000,C 90.000,E1 35.025} C_DIS
LIN {X -0.030,Y -227.214,Z 648.178,A 0.000,B 0.000,C 90.000,E1 32.054} C_DIS
LIN {X -0.020,Y -220.620,Z 648.161,A 0.000,B 0.000,C 90.000,E1 28.999} C_DIS
LIN {X 0.000,Y -214.904,Z 648.144,A 0.000,B 0.000,C 90.000,E1 25.899} C_DIS
LIN {X -0.007,Y -209.909,Z 648.126,A 0.000,B 0.000,C 90.000,E1 22.770} C_DIS
LIN {X 0.101,Y -204.736,Z 648.104,A 0.000,B 0.000,C 90.000,E1 18.779} C_DIS
LIN {X -0.085,Y -200.673,Z 648.082,A 0.000,B 0.000,C 90.000,E1 14.828} C_DIS
LIN {X -0.018,Y -197.207,Z 648.055,A 0.000,B 0.000,C 90.000,E1 9.962} C_DIS
LIN {X -0.035,Y -194.657,Z 648.015,A 0.000,B 0.000,C 90.000,E1 2.636} C_DIS
LIN {X 0.012,Y -196.374,Z 647.961,A 0.000,B 0.000,C 90.000,E1 352.996} C_DIS
LIN {X 0.018,Y -199.361,Z 647.934,A 0.000,B 0.000,C 90.000,E1 348.117} C_DIS
LIN {X -0.059,Y -202.931,Z 647.912,A 0.000,B 0.000,C 90.000,E1 344.102} C_DIS
LIN {X 0.073,Y -207.507,Z 647.889,A 0.000,B 0.000,C 90.000,E1 340.061} C_DIS
LIN {X 0.064,Y -212.936,Z 647.867,A 0.000,B 0.000,C 90.000,E1 336.102} C_DIS
LIN {X -0.106,Y -219.104,Z 647.846,A 0.000,B 0.000,C 90.000,E1 332.231} C_DIS
LIN {X 0.042,Y -225.958,Z 647.824,A 0.000,B 0.000,C 90.000,E1 328.329} C_DIS
LIN {X 0.012,Y -233.286,Z 647.803,A 0.000,B 0.000,C 90.000,E1 324.529} C_DIS
LIN {X -0.090,Y -241.231,Z 647.782,A 0.000,B 0.000,C 90.000,E1 320.803} C_DIS
LIN {X 0.115,Y -249.990,Z 647.762,A 0.000,B 0.000,C 90.000,E1 317.067} C_DIS
LIN {X 0.043,Y -259.759,Z 647.742,A 0.000,B 0.000,C 90.000,E1 313.461} C_DIS
LIN {X 0.107,Y -269.633,Z 647.724,A 0.000,B 0.000,C 90.000,E1 310.253} C_DIS
LIN {X 0.050,Y -282.132,Z 647.704,A 0.000,B 0.000,C 90.000,E1 306.790} C_DIS
LIN {X 0.183,Y -294.557,Z 647.687,A 0.000,B 0.000,C 90.000,E1 303.706} C_DIS
LIN {X 0.076,Y -309.902,Z 647.669,A 0.000,B 0.000,C 90.000,E1 300.413} C_DIS
LIN {X 0.059,Y -325.047,Z 647.653,A 0.000,B 0.000,C 90.000,E1 297.513} C_DIS
LIN {X -0.126,Y -338.925,Z 647.639,A 0.000,B 0.000,C 90.000,E1 295.027} C_DIS
LIN {X -0.089,Y -355.479,Z 647.624,A 0.000,B 0.000,C 90.000,E1 292.259} C_DIS
LIN {X -0.082,Y -371.135,Z 647.610,A 0.000,B 0.000,C 90.000,E1 289.866} C_DIS
LIN {X -0.050,Y -386.339,Z 647.599,A 0.000,B 0.000,C 90.000,E1 287.819} C_DIS
LIN {X -0.098,Y -404.973,Z 647.586,A 0.000,B 0.000,C 90.000,E1 285.552} C_DIS
LIN {X -0.003,Y -414.243,Z 647.580,A 0.000,B 0.000,C 90.000,E1 284.426} C_DIS
LIN {X 0.101,Y -427.505,Z 647.571,A 0.000,B 0.000,C 90.000,E1 282.771} C_DIS
LIN {X 0.146,Y -438.043,Z 647.564,A 0.000,B 0.000,C 90.000,E1 281.422} C_DIS
LIN {X -0.167,Y -448.019,Z 647.556,A 0.000,B 0.000,C 90.000,E1 280.141} C_DIS
LIN {X -0.157,Y -456.208,Z 647.550,A 0.000,B 0.000,C 90.000,E1 279.095} C_DIS
LIN {X -0.051,Y -464.807,Z 647.545,A 0.000,B 0.000,C 90.000,E1 278.049} C_DIS
LIN {X -0.158,Y -470.463,Z 647.540,A 0.000,B 0.000,C 90.000,E1 277.296} C_DIS
LIN {X -0.064,Y -473.782,Z 647.538,A 0.000,B 0.000,C 90.000,E1 276.777} C_DIS
LIN {X -0.144,Y -478.044,Z 647.533,A 0.000,B 0.000,C 90.000,E1 276.030} C_DIS
LIN {X -0.141,Y -481.508,Z 647.529,A 0.000,B 0.000,C 90.000,E1 275.277} C_DIS
LIN {X 0.022,Y -483.334,Z 647.526,A 0.000,B 0.000,C 90.000,E1 274.759} C_DIS
LIN {X 0.155,Y -484.790,Z 647.524,A 0.000,B 0.000,C 90.000,E1 274.245} C_DIS
LIN {X -0.150,Y -485.794,Z 647.521,A 0.000,B 0.000,C 90.000,E1 273.784} C_DIS
LIN {X 0.007,Y -486.452,Z 647.518,A 0.000,B 0.000,C 90.000,E1 273.269} C_DIS
LIN {X 0.198,Y -486.756,Z 647.515,A 0.000,B 0.000,C 90.000,E1 272.751} C_DIS
LIN {X -0.117,Y -486.807,Z 647.513,A 0.000,B 0.000,C 90.000,E1 272.293} C_DIS
LIN {X 0.073,Y -486.572,Z 647.510,A 0.000,B 0.000,C 90.000,E1 271.776} C_DIS
LIN {X -0.240,Y -485.962,Z 647.507,A 0.000,B 0.000,C 90.000,E1 271.318} C_DIS
LIN {X -0.067,Y -485.021,Z 647.504,A 0.000,B 0.000,C 90.000,E1 270.802} C_DIS
LIN {X 0.104,Y -483.586,Z 647.502,A 0.000,B 0.000,C 90.000,E1 270.286} C_DIS
LIN {X -0.213,Y -481.584,Z 647.499,A 0.000,B 0.000,C 90.000,E1 269.828} C_DIS
LIN {X -0.056,Y -478.890,Z 647.496,A 0.000,B 0.000,C 90.000,E1 269.312} C_DIS
LIN {X 0.080,Y -475.376,Z 647.493,A 0.000,B 0.000,C 90.000,E1 268.797} C_DIS
LIN {X -0.100,Y -473.311,Z 647.492,A 0.000,B 0.000,C 90.000,E1 268.568} C_DIS
LIN {X 0.020,Y -468.276,Z 647.489,A 0.000,B 0.000,C 90.000,E1 268.051} C_DIS
LIN {X -0.167,Y -465.278,Z 647.488,A 0.000,B 0.000,C 90.000,E1 267.822} C_DIS
LIN {X -0.049,Y -458.917,Z 647.485,A 0.000,B 0.000,C 90.000,E1 267.364} C_DIS
LIN {X 0.163,Y -451.996,Z 647.483,A 0.000,B 0.000,C 90.000,E1 266.963} C_DIS
LIN {X 0.071,Y -444.593,Z 647.482,A 0.000,B 0.000,C 90.000,E1 266.674} C_DIS
LIN {X 0.027,Y -436.604,Z 647.480,A 0.000,B 0.000,C 90.000,E1 266.445} C_DIS
LIN {X 0.023,Y -427.761,Z 647.479,A 0.000,B 0.000,C 90.000,E1 266.274} C_DIS
LIN {X -0.171,Y -419.377,Z 647.479,A 0.000,B 0.000,C 90.000,E1 266.216} C_DIS
LIN {X 0.042,Y -412.693,Z 647.479,A 0.000,B 0.000,C 90.000,E1 266.159} C_DIS
LIN {X -0.003,Y -180.928,Z 647.479,A 0.000,B 0.000,C 90.000,E1 266.159} C_DIS
LIN {X -0.093,Y -180.901,Z 647.474,A 0.000,B 0.000,C 90.000,E1 265.298} C_DIS
LIN {X 0.036,Y -180.230,Z 647.464,A 0.000,B 0.000,C 90.000,E1 263.571} C_DIS
LIN {X 0.052,Y -178.713,Z 647.441,A 0.000,B 0.000,C 90.000,E1 259.342} C_DIS
LIN {X -0.055,Y -175.762,Z 647.413,A 0.000,B 0.000,C 90.000,E1 254.283} C_DIS
LIN {X -0.005,Y -171.945,Z 647.384,A 0.000,B 0.000,C 90.000,E1 249.135} C_DIS
LIN {X -0.029,Y -171.330,Z 647.379,A 0.000,B 0.000,C 90.000,E1 248.284} C_DIS
LIN {X 0.024,Y -167.585,Z 647.355,A 0.000,B 0.000,C 90.000,E1 243.948} C_DIS
LIN {X -0.038,Y -166.222,Z 647.346,A 0.000,B 0.000,C 90.000,E1 242.231} C_DIS
LIN {X -0.049,Y -162.984,Z 647.326,A 0.000,B 0.000,C 90.000,E1 238.742} C_DIS
LIN {X -0.002,Y -160.900,Z 647.312,A 0.000,B 0.000,C 90.000,E1 236.087} C_DIS
LIN {X -0.023,Y -157.667,Z 647.292,A 0.000,B 0.000,C 90.000,E1 232.557} C_DIS
LIN {X -0.085,Y -155.705,Z 647.277,A 0.000,B 0.000,C 90.000,E1 229.908} C_DIS
LIN {X -0.030,Y -151.967,Z 647.252,A 0.000,B 0.000,C 90.000,E1 225.405} C_DIS
LIN {X -0.013,Y -150.210,Z 647.237,A 0.000,B 0.000,C 90.000,E1 222.690} C_DIS
LIN {X -0.089,Y -146.977,Z 647.212,A 0.000,B 0.000,C 90.000,E1 218.177} C_DIS
LIN {X 0.019,Y -145.563,Z 647.197,A 0.000,B 0.000,C 90.000,E1 215.391} C_DIS
LIN {X 0.019,Y -142.954,Z 647.171,A 0.000,B 0.000,C 90.000,E1 210.797} C_DIS
LIN {X -0.050,Y -141.580,Z 647.151,A 0.000,B 0.000,C 90.000,E1 207.129} C_DIS
LIN {X -0.002,Y -139.416,Z 647.115,A 0.000,B 0.000,C 90.000,E1 200.610} C_DIS
LIN {X 0.049,Y -139.140,Z 647.104,A 0.000,B 0.000,C 90.000,E1 198.725} C_DIS
LIN {X -0.060,Y -138.348,Z 647.057,A 0.000,B 0.000,C 90.000,E1 190.366} C_DIS
LIN {X 0.064,Y -139.492,Z 647.006,A 0.000,B 0.000,C 90.000,E1 180.974} C_DIS
LIN {X 0.005,Y -141.103,Z 646.975,A 0.000,B 0.000,C 90.000,E1 175.412} C_DIS
LIN {X -0.042,Y -142.482,Z 646.959,A 0.000,B 0.000,C 90.000,E1 172.648} C_DIS
LIN {X 0.048,Y -144.730,Z 646.933,A 0.000,B 0.000,C 90.000,E1 167.993} C_DIS
LIN {X -0.002,Y -147.335,Z 646.913,A 0.000,B 0.000,C 90.000,E1 164.338} C_DIS
LIN {X 0.063,Y -150.658,Z 646.888,A 0.000,B 0.000,C 90.000,E1 159.752} C_DIS
LIN {X -0.055,Y -154.136,Z 646.868,A 0.000,B 0.000,C 90.000,E1 156.177} C_DIS
LIN {X 0.007,Y -157.564,Z 646.848,A 0.000,B 0.000,C 90.000,E1 152.564} C_DIS
LIN {X 0.031,Y -161.808,Z 646.828,A 0.000,B 0.000,C 90.000,E1 148.997} C_DIS
LIN {X 0.051,Y -166.000,Z 646.808,A 0.000,B 0.000,C 90.000,E1 145.468} C_DIS
LIN {X 0.044,Y -170.998,Z 646.789,A 0.000,B 0.000,C 90.000,E1 141.984} C_DIS
LIN {X -0.041,Y -175.868,Z 646.770,A 0.000,B 0.000,C 90.000,E1 138.566} C_DIS
LIN {X -0.048,Y -181.472,Z 646.751,A 0.000,B 0.000,C 90.000,E1 135.162} C_DIS
LIN {X 0.089,Y -186.985,Z 646.732,A 0.000,B 0.000,C 90.000,E1 131.757} C_DIS
LIN {X 0.015,Y -191.049,Z 646.720,A 0.000,B 0.000,C 90.000,E1 129.600} C_DIS
LIN {X 0.155,Y -289.185,Z 646.720,A 0.000,B 0.000,C 90.000,E1 129.564} C_DIS
LIN {X -0.002,Y -290.651,Z 646.720,A 0.000,B 0.000,C 90.000,E1 129.564} C_DIS
LIN {X 0.069,Y -295.661,Z 646.718,A 0.000,B 0.000,C 90.000,E1 129.277} C_DIS
LIN {X 0.003,Y -298.904,Z 646.716,A 0.000,B 0.000,C 90.000,E1 128.955} C_DIS
LIN {X -0.050,Y -302.494,Z 646.713,A 0.000,B 0.000,C 90.000,E1 128.382} C_DIS
LIN {X 0.137,Y -303.923,Z 646.711,A 0.000,B 0.000,C 90.000,E1 128.016} C_DIS
LIN {X -0.103,Y -305.046,Z 646.709,A 0.000,B 0.000,C 90.000,E1 127.729} C_DIS
LIN {X 0.003,Y -315.606,Z 646.690,A 0.000,B 0.000,C 90.000,E1 124.119} C_DIS
LIN {X -0.124,Y -325.584,Z 646.674,A 0.000,B 0.000,C 90.000,E1 121.258} C_DIS
LIN {X -0.022,Y -336.884,Z 646.658,A 0.000,B 0.000,C 90.000,E1 118.409} C_DIS
LIN {X -0.083,Y -349.610,Z 646.642,A 0.000,B 0.000,C 90.000,E1 115.643} C_DIS
LIN {X 0.040,Y -362.210,Z 646.629,A 0.000,B 0.000,C 90.000,E1 113.206} C_DIS
LIN {X 0.010,Y -376.115,Z 646.616,A 0.000,B 0.000,C 90.000,E1 110.844} C_DIS
LIN {X -0.078,Y -391.425,Z 646.603,A 0.000,B 0.000,C 90.000,E1 108.544} C_DIS
LIN {X 0.103,Y -408.254,Z 646.590,A 0.000,B 0.000,C 90.000,E1 106.260} C_DIS
LIN {X 0.083,Y -426.723,Z 646.578,A 0.000,B 0.000,C 90.000,E1 104.064} C_DIS
LIN {X 0.173,Y -446.604,Z 646.567,A 0.000,B 0.000,C 90.000,E1 101.951} C_DIS
LIN {X 0.201,Y -467.089,Z 646.556,A 0.000,B 0.000,C 90.000,E1 100.018} C_DIS
LIN {X -0.228,Y -471.964,Z 646.553,A 0.000,B 0.000,C 90.000,E1 99.613} C_DIS
LIN {X 0.145,Y -473.813,Z 646.552,A 0.000,B 0.000,C 90.000,E1 99.321} C_DIS
LIN {X -0.024,Y -475.209,Z 646.551,A 0.000,B 0.000,C 90.000,E1 99.095} C_DIS
LIN {X 0.172,Y -477.037,Z 646.548,A 0.000,B 0.000,C 90.000,E1 98.568} C_DIS
LIN {X -0.170,Y -477.769,Z 646.545,A 0.000,B 0.000,C 90.000,E1 98.106} C_DIS
LIN {X -0.026,Y -477.528,Z 646.542,A 0.000,B 0.000,C 90.000,E1 97.587} C_DIS
LIN {X 0.124,Y -476.283,Z 646.539,A 0.000,B 0.000,C 90.000,E1 97.068} C_DIS
LIN {X -0.011,Y -475.223,Z 646.538,A 0.000,B 0.000,C 90.000,E1 96.834} C_DIS
LIN {X -0.200,Y -473.801,Z 646.537,A 0.000,B 0.000,C 90.000,E1 96.606} C_DIS
LIN {X -0.197,Y -456.592,Z 646.522,A 0.000,B 0.000,C 90.000,E1 94.069} C_DIS
LIN {X -0.023,Y -445.840,Z 646.512,A 0.000,B 0.000,C 90.000,E1 92.236} C_DIS
LIN {X 0.106,Y -434.330,Z 646.501,A 0.000,B 0.000,C 90.000,E1 90.115} C_DIS
LIN {X -0.007,Y -426.896,Z 646.493,A 0.000,B 0.000,C 90.000,E1 88.797} C_DIS
LIN {X -0.108,Y -417.588,Z 646.484,A 0.000,B 0.000,C 90.000,E1 87.192} C_DIS
LIN {X -0.174,Y -405.110,Z 646.472,A 0.000,B 0.000,C 90.000,E1 85.008} C_DIS
LIN {X -0.029,Y -391.453,Z 646.458,A 0.000,B 0.000,C 90.000,E1 82.470} C_DIS
LIN {X -0.135,Y -378.354,Z 646.444,A 0.000,B 0.000,C 90.000,E1 79.916} C_DIS
LIN {X -0.150,Y -367.094,Z 646.431,A 0.000,B 0.000,C 90.000,E1 77.589} C_DIS
LIN {X 0.181,Y -354.874,Z 646.416,A 0.000,B 0.000,C 90.000,E1 74.866} C_DIS
LIN {X -0.060,Y -343.406,Z 646.401,A 0.000,B 0.000,C 90.000,E1 72.181} C_DIS
LIN {X -0.035,Y -329.019,Z 646.380,A 0.000,B 0.000,C 90.000,E1 68.465} C_DIS
LIN {X -0.024,Y -316.079,Z 646.359,A 0.000,B 0.000,C 90.000,E1 64.665} C_DIS
LIN {X -0.007,Y -306.350,Z 646.341,A 0.000,B 0.000,C 90.000,E1 61.435} C_DIS
LIN {X 0.155,Y -297.434,Z 646.323,A 0.000,B 0.000,C 90.000,E1 58.122} C_DIS
LIN {X 0.011,Y -289.112,Z 646.305,A 0.000,B 0.000,C 90.000,E1 54.815} C_DIS
LIN {X 0.018,Y -282.689,Z 646.289,A 0.000,B 0.000,C 90.000,E1 52.110} C_DIS
LIN {X -0.026,Y -277.735,Z 646.278,A 0.000,B 0.000,C 90.000,E1 50.070} C_DIS
LIN {X -0.012,Y -274.201,Z 646.271,A 0.000,B 0.000,C 90.000,E1 48.690} C_DIS
LIN {X -0.038,Y -270.457,Z 646.263,A 0.000,B 0.000,C 90.000,E1 47.310} C_DIS
LIN {X 0.010,Y -264.407,Z 646.251,A 0.000,B 0.000,C 90.000,E1 45.202} C_DIS
LIN {X -0.053,Y -257.924,Z 646.239,A 0.000,B 0.000,C 90.000,E1 43.095} C_DIS
LIN {X -0.038,Y -251.270,Z 646.227,A 0.000,B 0.000,C 90.000,E1 40.943} C_DIS
LIN {X 0.044,Y -242.649,Z 646.211,A 0.000,B 0.000,C 90.000,E1 38.016} C_DIS
LIN {X -0.152,Y -234.636,Z 646.195,A 0.000,B 0.000,C 90.000,E1 35.105} C_DIS
LIN {X -0.094,Y -227.374,Z 646.178,A 0.000,B 0.000,C 90.000,E1 32.084} C_DIS
LIN {X 0.038,Y -220.781,Z 646.161,A 0.000,B 0.000,C 90.000,E1 28.999} C_DIS
LIN {X -0.033,Y -215.047,Z 646.144,A 0.000,B 0.000,C 90.000,E1 25.924} C_DIS
LIN {X 0.055,Y -210.039,Z 646.127,A 0.000,B 0.000,C 90.000,E1 22.770} C_DIS
LIN {X -0.029,Y -204.850,Z 646.105,A 0.000,B 0.000,C 90.000,E1 18.833} C_DIS
LIN {X -0.018,Y -200.776,Z 646.082,A 0.000,B 0.000,C 90.000,E1 14.828} C_DIS
LIN {X 0.051,Y -197.318,Z 646.055,A 0.000,B 0.000,C 90.000,E1 9.962} C_DIS
LIN {X 0.040,Y -194.747,Z 646.015,A 0.000,B 0.000,C 90.000,E1 2.636} C_DIS
LIN {X 0.015,Y -196.455,Z 645.961,A 0.000,B 0.000,C 90.000,E1 352.996} C_DIS
LIN {X 0.025,Y -199.429,Z 645.934,A 0.000,B 0.000,C 90.000,E1 348.117} C_DIS
LIN {X -0.049,Y -203.006,Z 645.912,A 0.000,B 0.000,C 90.000,E1 344.102} C_DIS
LIN {X 0.086,Y -207.571,Z 645.889,A 0.000,B 0.000,C 90.000,E1 340.061} C_DIS
LIN {X 0.078,Y -212.993,Z 645.867,A 0.000,B 0.000,C 90.000,E1 336.102} C_DIS
LIN {X -0.089,Y -219.159,Z 645.846,A 0.000,B 0.000,C 90.000,E1 332.231} C_DIS
LIN {X 0.061,Y -226.001,Z 645.824,A 0.000,B 0.000,C 90.000,E1 328.329} C_DIS
LIN {X 0.032,Y -233.311,Z 645.803,A 0.000,B 0.000,C 90.000,E1 324.529} C_DIS
LIN {X -0.068,Y -241.246,Z 645.782,A 0.000,B 0.000,C 90.000,E1 320.803} C_DIS
LIN {X -0.033,Y -249.977,Z 645.762,A 0.000,B 0.000,C 90.000,E1 317.106} C_DIS
LIN {X 0.067,Y -259.725,Z 645.742,A 0.000,B 0.000,C 90.000,E1 313.461} C_DIS
LIN {X -0.075,Y -269.571,Z 645.724,A 0.000,B 0.000,C 90.000,E1 310.297} C_DIS
LIN {X 0.073,Y -282.055,Z 645.704,A 0.000,B 0.000,C 90.000,E1 306.790} C_DIS
LIN {X -0.049,Y -295.958,Z 645.686,A 0.000,B 0.000,C 90.000,E1 303.420} C_DIS
LIN {X -0.129,Y -311.447,Z 645.667,A 0.000,B 0.000,C 90.000,E1 300.129} C_DIS
LIN {X 0.077,Y -324.950,Z 645.653,A 0.000,B 0.000,C 90.000,E1 297.513} C_DIS
LIN {X -0.110,Y -338.822,Z 645.639,A 0.000,B 0.000,C 90.000,E1 295.027} C_DIS
LIN {X -0.075,Y -355.376,Z 645.624,A 0.000,B 0.000,C 90.000,E1 292.259} C_DIS
LIN {X -0.069,Y -371.055,Z 645.610,A 0.000,B 0.000,C 90.000,E1 289.866} C_DIS
LIN {X -0.038,Y -386.261,Z 645.599,A 0.000,B 0.000,C 90.000,E1 287.819} C_DIS
LIN {X -0.088,Y -404.889,Z 645.586,A 0.000,B 0.000,C 90.000,E1 285.552} C_DIS
LIN {X 0.007,Y -414.160,Z 645.580,A 0.000,B 0.000,C 90.000,E1 284.426} C_DIS
LIN {X -0.050,Y -425.229,Z 645.573,A 0.000,B 0.000,C 90.000,E1 283.063} C_DIS
LIN {X -0.036,Y -435.875,Z 645.565,A 0.000,B 0.000,C 90.000,E1 281.715} C_DIS
LIN {X -0.088,Y -444.021,Z 645.559,A 0.000,B 0.000,C 90.000,E1 280.658} C_DIS
LIN {X 0.113,Y -454.028,Z 645.552,A 0.000,B 0.000,C 90.000,E1 279.321} C_DIS
LIN {X -0.046,Y -464.735,Z 645.545,A 0.000,B 0.000,C 90.000,E1 278.049} C_DIS
LIN {X -0.154,Y -470.367,Z 645.540,A 0.000,B 0.000,C 90.000,E1 277.296} C_DIS
LIN {X -0.061,Y -473.669,Z 645.538,A 0.000,B 0.000,C 90.000,E1 276.777} C_DIS
LIN {X -0.141,Y -477.939,Z 645.533,A 0.000,B 0.000,C 90.000,E1 276.030} C_DIS
LIN {X -0.139,Y -481.421,Z 645.529,A 0.000,B 0.000,C 90.000,E1 275.277} C_DIS
LIN {X 0.024,Y -483.258,Z 645.526,A 0.000,B 0.000,C 90.000,E1 274.759} C_DIS
LIN {X 0.155,Y -484.687,Z 645.524,A 0.000,B 0.000,C 90.000,E1 274.245} C_DIS
LIN {X -0.150,Y -485.720,Z 645.521,A 0.000,B 0.000,C 90.000,E1 273.784} C_DIS
LIN {X 0.007,Y -486.365,Z 645.518,A 0.000,B 0.000,C 90.000,E1 273.269} C_DIS
LIN {X 0.197,Y -486.677,Z 645.515,A 0.000,B 0.000,C 90.000,E1 272.751} C_DIS
LIN {X -0.119,Y -486.743,Z 645.513,A 0.000,B 0.000,C 90.000,E1 272.293} C_DIS
LIN {X 0.071,Y -486.520,Z 645.510,A 0.000,B 0.000,C 90.000,E1 271.776} C_DIS
LIN {X 0.244,Y -485.932,Z 645.507,A 0.000,B 0.000,C 90.000,E1 271.260} C_DIS
LIN {X -0.068,Y -484.999,Z 645.504,A 0.000,B 0.000,C 90.000,E1 270.802} C_DIS
LIN {X 0.101,Y -483.527,Z 645.502,A 0.000,B 0.000,C 90.000,E1 270.286} C_DIS
LIN {X -0.215,Y -481.573,Z 645.499,A 0.000,B 0.000,C 90.000,E1 269.828} C_DIS
LIN {X -0.059,Y -478.888,Z 645.496,A 0.000,B 0.000,C 90.000,E1 269.312} C_DIS
LIN {X 0.076,Y -475.409,Z 645.493,A 0.000,B 0.000,C 90.000,E1 268.797} C_DIS
LIN {X 0.191,Y -470.936,Z 645.491,A 0.000,B 0.000,C 90.000,E1 268.282} C_DIS
LIN {X -0.169,Y -465.284,Z 645.488,A 0.000,B 0.000,C 90.000,E1 267.822} C_DIS
LIN {X -0.118,Y -462.322,Z 645.487,A 0.000,B 0.000,C 90.000,E1 267.593} C_DIS
LIN {X -0.069,Y -458.940,Z 645.485,A 0.000,B 0.000,C 90.000,E1 267.364} C_DIS
LIN {X -0.185,Y -455.697,Z 645.484,A 0.000,B 0.000,C 90.000,E1 267.192} C_DIS
LIN {X -0.092,Y -448.599,Z 645.482,A 0.000,B 0.000,C 90.000,E1 266.846} C_DIS
LIN {X 0.068,Y -440.986,Z 645.481,A 0.000,B 0.000,C 90.000,E1 266.560} C_DIS
LIN {X -0.175,Y -432.883,Z 645.480,A 0.000,B 0.000,C 90.000,E1 266.388} C_DIS
LIN {X 0.043,Y -423.167,Z 645.479,A 0.000,B 0.000,C 90.000,E1 266.216} C_DIS
LIN {X 0.002,Y -410.891,Z 645.479,A 0.000,B 0.000,C 90.000,E1 266.159} C_DIS
LIN {X -0.021,Y -180.927,Z 645.479,A 0.000,B 0.000,C 90.000,E1 266.159} C_DIS
LIN {X -0.093,Y -180.901,Z 645.474,A 0.000,B 0.000,C 90.000,E1 265.298} C_DIS
LIN {X 0.037,Y -180.230,Z 645.464,A 0.000,B 0.000,C 90.000,E1 263.571} C_DIS
LIN {X 0.053,Y -178.712,Z 645.441,A 0.000,B 0.000,C 90.000,E1 259.342} C_DIS
LIN {X -0.054,Y -175.761,Z 645.413,A 0.000,B 0.000,C 90.000,E1 254.283} C_DIS
LIN {X -0.004,Y -171.945,Z 645.384,A 0.000,B 0.000,C 90.000,E1 249.135} C_DIS
LIN {X -0.028,Y -171.331,Z 645.379,A 0.000,B 0.000,C 90.000,E1 248.284} C_DIS
LIN {X 0.024,Y -167.586,Z 645.355,A 0.000,B 0.000,C 90.000,E1 243.948} C_DIS
LIN {X -0.036,Y -166.222,Z 645.346,A 0.000,B 0.000,C 90.000,E1 242.231} C_DIS
LIN {X -0.047,Y -162.984,Z 645.326,A 0.000,B 0.000,C 90.000,E1 238.742} C_DIS
LIN {X -0.001,Y -160.900,Z 645.312,A 0.000,B 0.000,C 90.000,E1 236.087} C_DIS
LIN {X -0.023,Y -157.667,Z 645.292,A 0.000,B 0.000,C 90.000,E1 232.557} C_DIS
LIN {X -0.084,Y -155.706,Z 645.277,A 0.000,B 0.000,C 90.000,E1 229.908} C_DIS
LIN {X -0.030,Y -151.968,Z 645.252,A 0.000,B 0.000,C 90.000,E1 225.405} C_DIS
LIN {X -0.013,Y -150.210,Z 645.237,A 0.000,B 0.000,C 90.000,E1 222.690} C_DIS
LIN {X -0.089,Y -146.976,Z 645.212,A 0.000,B 0.000,C 90.000,E1 218.177} C_DIS
LIN {X 0.021,Y -145.562,Z 645.197,A 0.000,B 0.000,C 90.000,E1 215.391} C_DIS
LIN {X 0.020,Y -142.954,Z 645.171,A 0.000,B 0.000,C 90.000,E1 210.797} C_DIS
LIN {X -0.050,Y -141.580,Z 645.151,A 0.000,B 0.000,C 90.000,E1 207.129} C_DIS
LIN {X -0.002,Y -139.416,Z 645.115,A 0.000,B 0.000,C 90.000,E1 200.610} C_DIS
LIN {X 0.050,Y -139.141,Z 645.104,A 0.000,B 0.000,C 90.000,E1 198.725} C_DIS
LIN {X -0.059,Y -138.348,Z 645.057,A 0.000,B 0.000,C 90.000,E1 190.366} C_DIS
LIN {X 0.065,Y -139.492,Z 645.006,A 0.000,B 0.000,C 90.000,E1 180.974} C_DIS
LIN {X 0.006,Y -141.103,Z 644.975,A 0.000,B 0.000,C 90.000,E1 175.412} C_DIS
LIN {X -0.041,Y -142.482,Z 644.959,A 0.000,B 0.000,C 90.000,E1 172.648} C_DIS
LIN {X 0.048,Y -144.730,Z 644.933,A 0.000,B 0.000,C 90.000,E1 167.993} C_DIS
LIN {X -0.001,Y -147.335,Z 644.913,A 0.000,B 0.000,C 90.000,E1 164.338} C_DIS
LIN {X 0.064,Y -150.658,Z 644.888,A 0.000,B 0.000,C 90.000,E1 159.752} C_DIS
LIN {X -0.055,Y -154.136,Z 644.868,A 0.000,B 0.000,C 90.000,E1 156.177} C_DIS
LIN {X 0.007,Y -157.564,Z 644.848,A 0.000,B 0.000,C 90.000,E1 152.564} C_DIS
LIN {X 0.032,Y -161.807,Z 644.828,A 0.000,B 0.000,C 90.000,E1 148.997} C_DIS
LIN {X 0.052,Y -165.999,Z 644.808,A 0.000,B 0.000,C 90.000,E1 145.468} C_DIS
LIN {X 0.044,Y -170.997,Z 644.789,A 0.000,B 0.000,C 90.000,E1 141.984} C_DIS
LIN {X -0.040,Y -175.867,Z 644.770,A 0.000,B 0.000,C 90.000,E1 138.566} C_DIS
LIN {X -0.047,Y -181.472,Z 644.751,A 0.000,B 0.000,C 90.000,E1 135.162} C_DIS
LIN {X 0.090,Y -186.984,Z 644.732,A 0.000,B 0.000,C 90.000,E1 131.757} C_DIS
LIN {X -0.110,Y -191.038,Z 644.720,A 0.000,B 0.000,C 90.000,E1 129.644} C_DIS
LIN {X 0.024,Y -288.486,Z 644.720,A 0.000,B 0.000,C 90.000,E1 129.600} C_DIS
LIN {X 0.048,Y -293.409,Z 644.719,A 0.000,B 0.000,C 90.000,E1 129.439} C_DIS
LIN {X 0.070,Y -295.671,Z 644.718,A 0.000,B 0.000,C 90.000,E1 129.277} C_DIS
LIN {X -0.010,Y -299.528,Z 644.716,A 0.000,B 0.000,C 90.000,E1 128.874} C_DIS
LIN {X 0.140,Y -301.453,Z 644.714,A 0.000,B 0.000,C 90.000,E1 128.543} C_DIS
LIN {X 0.058,Y -302.971,Z 644.713,A 0.000,B 0.000,C 90.000,E1 128.257} C_DIS
LIN {X 0.014,Y -304.285,Z 644.711,A 0.000,B 0.000,C 90.000,E1 127.935} C_DIS
LIN {X 0.006,Y -307.112,Z 644.705,A 0.000,B 0.000,C 90.000,E1 126.950} C_DIS
LIN {X -0.051,Y -316.960,Z 644.687,A 0.000,B 0.000,C 90.000,E1 123.706} C_DIS
LIN {X 0.141,Y -327.122,Z 644.671,A 0.000,B 0.000,C 90.000,E1 120.797} C_DIS
LIN {X 0.134,Y -338.626,Z 644.656,A 0.000,B 0.000,C 90.000,E1 117.975} C_DIS
LIN {X 0.142,Y -351.565,Z 644.640,A 0.000,B 0.000,C 90.000,E1 115.207} C_DIS
LIN {X -0.007,Y -364.372,Z 644.627,A 0.000,B 0.000,C 90.000,E1 112.823} C_DIS
LIN {X -0.126,Y -378.498,Z 644.614,A 0.000,B 0.000,C 90.000,E1 110.482} C_DIS
LIN {X -0.157,Y -394.049,Z 644.601,A 0.000,B 0.000,C 90.000,E1 108.181} C_DIS
LIN {X 0.086,Y -411.138,Z 644.588,A 0.000,B 0.000,C 90.000,E1 105.898} C_DIS
LIN {X 0.031,Y -429.887,Z 644.576,A 0.000,B 0.000,C 90.000,E1 103.716} C_DIS
LIN {X -0.101,Y -449.889,Z 644.565,A 0.000,B 0.000,C 90.000,E1 101.658} C_DIS
LIN {X 0.133,Y -470.445,Z 644.554,A 0.000,B 0.000,C 90.000,E1 99.726} C_DIS
LIN {X 0.118,Y -472.556,Z 644.553,A 0.000,B 0.000,C 90.000,E1 99.500} C_DIS
LIN {X -0.027,Y -474.317,Z 644.551,A 0.000,B 0.000,C 90.000,E1 99.265} C_DIS
LIN {X -0.174,Y -475.640,Z 644.550,A 0.000,B 0.000,C 90.000,E1 99.029} C_DIS
LIN {X -0.050,Y -477.291,Z 644.547,A 0.000,B 0.000,C 90.000,E1 98.511} C_DIS
LIN {X 0.085,Y -477.877,Z 644.544,A 0.000,B 0.000,C 90.000,E1 97.992} C_DIS
LIN {X -0.242,Y -477.495,Z 644.542,A 0.000,B 0.000,C 90.000,E1 97.530} C_DIS
LIN {X -0.033,Y -476.089,Z 644.539,A 0.000,B 0.000,C 90.000,E1 97.004} C_DIS
LIN {X -0.224,Y -474.932,Z 644.537,A 0.000,B 0.000,C 90.000,E1 96.777} C_DIS
LIN {X -0.085,Y -471.596,Z 644.535,A 0.000,B 0.000,C 90.000,E1 96.258} C_DIS
LIN {X 0.044,Y -456.176,Z 644.522,A 0.000,B 0.000,C 90.000,E1 93.955} C_DIS
LIN {X 0.205,Y -445.463,Z 644.512,A 0.000,B 0.000,C 90.000,E1 92.121} C_DIS
LIN {X -0.113,Y -433.957,Z 644.500,A 0.000,B 0.000,C 90.000,E1 90.057} C_DIS
LIN {X 0.197,Y -426.509,Z 644.493,A 0.000,B 0.000,C 90.000,E1 88.682} C_DIS
LIN {X 0.085,Y -417.193,Z 644.484,A 0.000,B 0.000,C 90.000,E1 87.078} C_DIS
LIN {X 0.002,Y -404.721,Z 644.472,A 0.000,B 0.000,C 90.000,E1 84.894} C_DIS
LIN {X 0.187,Y -389.596,Z 644.456,A 0.000,B 0.000,C 90.000,E1 82.064} C_DIS
LIN {X 0.039,Y -375.169,Z 644.440,A 0.000,B 0.000,C 90.000,E1 79.218} C_DIS
LIN {X 0.015,Y -364.016,Z 644.427,A 0.000,B 0.000,C 90.000,E1 76.881} C_DIS
LIN {X -0.183,Y -348.173,Z 644.407,A 0.000,B 0.000,C 90.000,E1 73.323} C_DIS
LIN {X -0.074,Y -335.802,Z 644.390,A 0.000,B 0.000,C 90.000,E1 70.242} C_DIS
LIN {X -0.084,Y -322.196,Z 644.369,A 0.000,B 0.000,C 90.000,E1 66.485} C_DIS
LIN {X 0.092,Y -310.026,Z 644.348,A 0.000,B 0.000,C 90.000,E1 62.615} C_DIS
LIN {X -0.047,Y -300.822,Z 644.330,A 0.000,B 0.000,C 90.000,E1 59.380} C_DIS
LIN {X -0.155,Y -292.302,Z 644.311,A 0.000,B 0.000,C 90.000,E1 56.087} C_DIS
LIN {X 0.162,Y -285.785,Z 644.297,A 0.000,B 0.000,C 90.000,E1 53.336} C_DIS
LIN {X 0.001,Y -280.999,Z 644.285,A 0.000,B 0.000,C 90.000,E1 51.331} C_DIS
LIN {X -0.113,Y -275.902,Z 644.274,A 0.000,B 0.000,C 90.000,E1 49.299} C_DIS
LIN {X -0.117,Y -272.258,Z 644.266,A 0.000,B 0.000,C 90.000,E1 47.919} C_DIS
LIN {X 0.017,Y -268.364,Z 644.258,A 0.000,B 0.000,C 90.000,E1 46.500} C_DIS
LIN {X 0.100,Y -264.277,Z 644.251,A 0.000,B 0.000,C 90.000,E1 45.081} C_DIS
LIN {X 0.026,Y -257.748,Z 644.239,A 0.000,B 0.000,C 90.000,E1 42.975} C_DIS
LIN {X 0.041,Y -249.965,Z 644.225,A 0.000,B 0.000,C 90.000,E1 40.458} C_DIS
LIN {X 0.107,Y -240.435,Z 644.207,A 0.000,B 0.000,C 90.000,E1 37.156} C_DIS
LIN {X 0.045,Y -232.600,Z 644.190,A 0.000,B 0.000,C 90.000,E1 34.199} C_DIS
LIN {X -0.075,Y -225.533,Z 644.173,A 0.000,B 0.000,C 90.000,E1 31.209} C_DIS
LIN {X 0.094,Y -219.170,Z 644.156,A 0.000,B 0.000,C 90.000,E1 28.103} C_DIS
LIN {X -0.014,Y -213.648,Z 644.139,A 0.000,B 0.000,C 90.000,E1 25.027} C_DIS
LIN {X -0.020,Y -207.762,Z 644.117,A 0.000,B 0.000,C 90.000,E1 21.099} C_DIS
LIN {X 0.075,Y -203.060,Z 644.095,A 0.000,B 0.000,C 90.000,E1 17.094} C_DIS
LIN {X -0.072,Y -199.463,Z 644.073,A 0.000,B 0.000,C 90.000,E1 13.119} C_DIS
LIN {X 0.057,Y -196.141,Z 644.041,A 0.000,B 0.000,C 90.000,E1 7.409} C_DIS
LIN {X 0.005,Y -196.939,Z 643.957,A 0.000,B 0.000,C 90.000,E1 352.186} C_DIS
LIN {X 0.069,Y -200.147,Z 643.930,A 0.000,B 0.000,C 90.000,E1 347.297} C_DIS
LIN {X 0.069,Y -203.919,Z 643.907,A 0.000,B 0.000,C 90.000,E1 343.268} C_DIS
LIN {X 0.107,Y -208.654,Z 643.885,A 0.000,B 0.000,C 90.000,E1 339.263} C_DIS
LIN {X -0.065,Y -214.235,Z 643.863,A 0.000,B 0.000,C 90.000,E1 335.357} C_DIS
LIN {X -0.001,Y -220.512,Z 643.841,A 0.000,B 0.000,C 90.000,E1 331.435} C_DIS
LIN {X 0.006,Y -227.449,Z 643.820,A 0.000,B 0.000,C 90.000,E1 327.582} C_DIS
LIN {X 0.016,Y -234.869,Z 643.799,A 0.000,B 0.000,C 90.000,E1 323.783} C_DIS
LIN {X -0.085,Y -242.919,Z 643.778,A 0.000,B 0.000,C 90.000,E1 320.070} C_DIS
LIN {X -0.017,Y -251.843,Z 643.758,A 0.000,B 0.000,C 90.000,E1 316.377} C_DIS
LIN {X -0.027,Y -261.764,Z 643.738,A 0.000,B 0.000,C 90.000,E1 312.771} C_DIS
LIN {X 0.096,Y -271.921,Z 643.720,A 0.000,B 0.000,C 90.000,E1 309.564} C_DIS
LIN {X 0.038,Y -283.322,Z 643.703,A 0.000,B 0.000,C 90.000,E1 306.457} C_DIS
LIN {X -0.029,Y -295.887,Z 643.686,A 0.000,B 0.000,C 90.000,E1 303.420} C_DIS
LIN {X -0.111,Y -311.364,Z 643.667,A 0.000,B 0.000,C 90.000,E1 300.129} C_DIS
LIN {X 0.094,Y -324.856,Z 643.653,A 0.000,B 0.000,C 90.000,E1 297.513} C_DIS
LIN {X -0.076,Y -336.946,Z 643.641,A 0.000,B 0.000,C 90.000,E1 295.335} C_DIS
LIN {X -0.092,Y -353.370,Z 643.625,A 0.000,B 0.000,C 90.000,E1 292.567} C_DIS
LIN {X -0.057,Y -370.977,Z 643.610,A 0.000,B 0.000,C 90.000,E1 289.866} C_DIS
LIN {X -0.029,Y -386.188,Z 643.599,A 0.000,B 0.000,C 90.000,E1 287.819} C_DIS
LIN {X -0.158,Y -402.459,Z 643.588,A 0.000,B 0.000,C 90.000,E1 285.843} C_DIS
LIN {X -0.098,Y -411.802,Z 643.582,A 0.000,B 0.000,C 90.000,E1 284.717} C_DIS
LIN {X -0.187,Y -422.949,Z 643.574,A 0.000,B 0.000,C 90.000,E1 283.355} C_DIS
LIN {X -0.219,Y -433.709,Z 643.567,A 0.000,B 0.000,C 90.000,E1 282.007} C_DIS
LIN {X 0.135,Y -441.956,Z 643.561,A 0.000,B 0.000,C 90.000,E1 280.894} C_DIS
LIN {X -0.148,Y -456.106,Z 643.550,A 0.000,B 0.000,C 90.000,E1 279.095} C_DIS
LIN {X -0.043,Y -464.597,Z 643.545,A 0.000,B 0.000,C 90.000,E1 278.049} C_DIS
LIN {X 0.015,Y -468.471,Z 643.542,A 0.000,B 0.000,C 90.000,E1 277.530} C_DIS
LIN {X -0.059,Y -473.554,Z 643.538,A 0.000,B 0.000,C 90.000,E1 276.777} C_DIS
LIN {X -0.140,Y -477.845,Z 643.533,A 0.000,B 0.000,C 90.000,E1 276.030} C_DIS
LIN {X 0.002,Y -480.231,Z 643.531,A 0.000,B 0.000,C 90.000,E1 275.511} C_DIS
LIN {X -0.139,Y -481.316,Z 643.529,A 0.000,B 0.000,C 90.000,E1 275.277} C_DIS
LIN {X 0.022,Y -483.129,Z 643.526,A 0.000,B 0.000,C 90.000,E1 274.759} C_DIS
LIN {X 0.153,Y -484.591,Z 643.524,A 0.000,B 0.000,C 90.000,E1 274.245} C_DIS
LIN {X -0.152,Y -485.587,Z 643.521,A 0.000,B 0.000,C 90.000,E1 273.784} C_DIS
LIN {X 0.004,Y -486.229,Z 643.518,A 0.000,B 0.000,C 90.000,E1 273.269} C_DIS
LIN {X 0.194,Y -486.585,Z 643.515,A 0.000,B 0.000,C 90.000,E1 272.751} C_DIS
LIN {X -0.123,Y -486.684,Z 643.513,A 0.000,B 0.000,C 90.000,E1 272.293} C_DIS
LIN {X 0.066,Y -486.458,Z 643.510,A 0.000,B 0.000,C 90.000,E1 271.776} C_DIS
LIN {X 0.239,Y -485.905,Z 643.507,A 0.000,B 0.000,C 90.000,E1 271.260} C_DIS
LIN {X -0.074,Y -484.963,Z 643.504,A 0.000,B 0.000,C 90.000,E1 270.802} C_DIS
LIN {X 0.096,Y -483.538,Z 643.502,A 0.000,B 0.000,C 90.000,E1 270.286} C_DIS
LIN {X -0.221,Y -481.567,Z 643.499,A 0.000,B 0.000,C 90.000,E1 269.828} C_DIS
LIN {X -0.065,Y -478.863,Z 643.496,A 0.000,B 0.000,C 90.000,E1 269.312} C_DIS
LIN {X 0.070,Y -475.391,Z 643.493,A 0.000,B 0.000,C 90.000,E1 268.797} C_DIS
LIN {X -0.108,Y -473.312,Z 643.492,A 0.000,B 0.000,C 90.000,E1 268.568} C_DIS
LIN {X 0.011,Y -468.311,Z 643.489,A 0.000,B 0.000,C 90.000,E1 268.051} C_DIS
LIN {X -0.118,Y -462.362,Z 643.487,A 0.000,B 0.000,C 90.000,E1 267.593} C_DIS
LIN {X -0.061,Y -459.005,Z 643.485,A 0.000,B 0.000,C 90.000,E1 267.364} C_DIS
LIN {X -0.181,Y -455.777,Z 643.484,A 0.000,B 0.000,C 90.000,E1 267.192} C_DIS
LIN {X -0.097,Y -448.662,Z 643.482,A 0.000,B 0.000,C 90.000,E1 266.846} C_DIS
LIN {X 0.066,Y -441.027,Z 643.481,A 0.000,B 0.000,C 90.000,E1 266.560} C_DIS
LIN {X -0.169,Y -432.890,Z 643.480,A 0.000,B 0.000,C 90.000,E1 266.388} C_DIS
LIN {X 0.040,Y -428.059,Z 643.479,A 0.000,B 0.000,C 90.000,E1 266.274} C_DIS
LIN {X -0.179,Y -419.401,Z 643.479,A 0.000,B 0.000,C 90.000,E1 266.216} C_DIS
LIN {X -0.019,Y -409.883,Z 643.479,A 0.000,B 0.000,C 90.000,E1 266.159} C_DIS
LIN {X -0.029,Y -180.927,Z 643.479,A 0.000,B 0.000,C 90.000,E1 266.159} C_DIS
LIN {X -0.092,Y -180.902,Z 643.474,A 0.000,B 0.000,C 90.000,E1 265.298} C_DIS
LIN {X 0.037,Y -180.230,Z 643.464,A 0.000,B 0.000,C 90.000,E1 263.571} C_DIS
LIN {X 0.053,Y -178.713,Z 643.441,A 0.000,B 0.000,C 90.000,E1 259.342} C_DIS
LIN {X -0.054,Y -175.761,Z 643.413,A 0.000,B 0.000,C 90.000,E1 254.283} C_DIS
LIN {X -0.004,Y -171.945,Z 643.384,A 0.000,B 0.000,C 90.000,E1 249.135} C_DIS
LIN {X -0.028,Y -171.331,Z 643.379,A 0.000,B 0.000,C 90.000,E1 248.284} C_DIS
LIN {X 0.025,Y -167.586,Z 643.355,A 0.000,B 0.000,C 90.000,E1 243.948} C_DIS
LIN {X -0.036,Y -166.222,Z 643.346,A 0.000,B 0.000,C 90.000,E1 242.231} C_DIS
LIN {X -0.047,Y -162.984,Z 643.326,A 0.000,B 0.000,C 90.000,E1 238.742} C_DIS
LIN {X -0.001,Y -160.900,Z 643.312,A 0.000,B 0.000,C 90.000,E1 236.087} C_DIS
LIN {X -0.023,Y -157.668,Z 643.292,A 0.000,B 0.000,C 90.000,E1 232.557} C_DIS
LIN {X -0.084,Y -155.705,Z 643.277,A 0.000,B 0.000,C 90.000,E1 229.908} C_DIS
LIN {X -0.030,Y -151.968,Z 643.252,A 0.000,B 0.000,C 90.000,E1 225.405} C_DIS
LIN {X -0.012,Y -150.210,Z 643.237,A 0.000,B 0.000,C 90.000,E1 222.690} C_DIS
LIN {X -0.088,Y -146.976,Z 643.212,A 0.000,B 0.000,C 90.000,E1 218.177} C_DIS
LIN {X 0.021,Y -145.562,Z 643.197,A 0.000,B 0.000,C 90.000,E1 215.391} C_DIS
LIN {X 0.020,Y -142.954,Z 643.171,A 0.000,B 0.000,C 90.000,E1 210.797} C_DIS
LIN {X -0.049,Y -141.580,Z 643.151,A 0.000,B 0.000,C 90.000,E1 207.129} C_DIS
LIN {X -0.002,Y -139.416,Z 643.115,A 0.000,B 0.000,C 90.000,E1 200.610} C_DIS
LIN {X 0.050,Y -139.141,Z 643.104,A 0.000,B 0.000,C 90.000,E1 198.725} C_DIS
LIN {X -0.058,Y -138.348,Z 643.057,A 0.000,B 0.000,C 90.000,E1 190.366} C_DIS
LIN {X 0.066,Y -139.491,Z 643.006,A 0.000,B 0.000,C 90.000,E1 180.974} C_DIS
LIN {X 0.007,Y -141.103,Z 642.975,A 0.000,B 0.000,C 90.000,E1 175.412} C_DIS
LIN {X -0.040,Y -142.482,Z 642.959,A 0.000,B 0.000,C 90.000,E1 172.648} C_DIS
LIN {X 0.049,Y -144.730,Z 642.933,A 0.000,B 0.000,C 90.000,E1 167.993} C_DIS
LIN {X 0.000,Y -147.334,Z 642.913,A 0.000,B 0.000,C 90.000,E1 164.338} C_DIS
LIN {X 0.065,Y -150.657,Z 642.888,A 0.000,B 0.000,C 90.000,E1 159.752} C_DIS
LIN {X -0.055,Y -154.136,Z 642.868,A 0.000,B 0.000,C 90.000,E1 156.177} C_DIS
LIN {X 0.008,Y -157.564,Z 642.848,A 0.000,B 0.000,C 90.000,E1 152.564} C_DIS
LIN {X 0.033,Y -161.807,Z 642.828,A 0.000,B 0.000,C 90.000,E1 148.997} C_DIS
LIN {X 0.052,Y -165.999,Z 642.808,A 0.000,B 0.000,C 90.000,E1 145.468} C_DIS
LIN {X 0.045,Y -170.998,Z 642.789,A 0.000,B 0.000,C 90.000,E1 141.984} C_DIS
LIN {X -0.039,Y -175.867,Z 642.770,A 0.000,B 0.000,C 90.000,E1 138.566} C_DIS
LIN {X -0.046,Y -181.472,Z 642.751,A 0.000,B 0.000,C 90.000,E1 135.162} C_DIS
LIN {X 0.091,Y -186.985,Z 642.732,A 0.000,B 0.000,C 90.000,E1 131.757} C_DIS
LIN {X 0.017,Y -191.047,Z 642.720,A 0.000,B 0.000,C 90.000,E1 129.600} C_DIS
LIN {X 0.157,Y -289.133,Z 642.720,A 0.000,B 0.000,C 90.000,E1 129.564} C_DIS
LIN {X -0.001,Y -290.607,Z 642.720,A 0.000,B 0.000,C 90.000,E1 129.564} C_DIS
LIN {X 0.071,Y -295.619,Z 642.718,A 0.000,B 0.000,C 90.000,E1 129.277} C_DIS
LIN {X 0.007,Y -298.861,Z 642.716,A 0.000,B 0.000,C 90.000,E1 128.955} C_DIS
LIN {X -0.046,Y -302.451,Z 642.713,A 0.000,B 0.000,C 90.000,E1 128.382} C_DIS
LIN {X 0.142,Y -303.880,Z 642.711,A 0.000,B 0.000,C 90.000,E1 128.016} C_DIS
LIN {X -0.099,Y -305.003,Z 642.710,A 0.000,B 0.000,C 90.000,E1 127.729} C_DIS
LIN {X 0.007,Y -315.562,Z 642.690,A 0.000,B 0.000,C 90.000,E1 124.119} C_DIS
LIN {X -0.121,Y -325.540,Z 642.674,A 0.000,B 0.000,C 90.000,E1 121.258} C_DIS
LIN {X -0.021,Y -336.839,Z 642.658,A 0.000,B 0.000,C 90.000,E1 118.409} C_DIS
LIN {X -0.083,Y -349.565,Z 642.642,A 0.000,B 0.000,C 90.000,E1 115.643} C_DIS
LIN {X 0.038,Y -362.164,Z 642.629,A 0.000,B 0.000,C 90.000,E1 113.206} C_DIS
LIN {X 0.006,Y -376.069,Z 642.616,A 0.000,B 0.000,C 90.000,E1 110.844} C_DIS
LIN {X -0.083,Y -391.380,Z 642.603,A 0.000,B 0.000,C 90.000,E1 108.544} C_DIS
LIN {X 0.097,Y -408.207,Z 642.590,A 0.000,B 0.000,C 90.000,E1 106.260} C_DIS
LIN {X 0.076,Y -426.676,Z 642.578,A 0.000,B 0.000,C 90.000,E1 104.064} C_DIS
LIN {X 0.164,Y -446.558,Z 642.567,A 0.000,B 0.000,C 90.000,E1 101.951} C_DIS
LIN {X 0.191,Y -467.042,Z 642.556,A 0.000,B 0.000,C 90.000,E1 100.018} C_DIS
LIN {X 0.228,Y -471.969,Z 642.553,A 0.000,B 0.000,C 90.000,E1 99.557} C_DIS
LIN {X 0.161,Y -473.837,Z 642.552,A 0.000,B 0.000,C 90.000,E1 99.321} C_DIS
LIN {X 0.020,Y -475.253,Z 642.551,A 0.000,B 0.000,C 90.000,E1 99.095} C_DIS
LIN {X 0.216,Y -477.143,Z 642.548,A 0.000,B 0.000,C 90.000,E1 98.568} C_DIS
LIN {X -0.125,Y -477.925,Z 642.545,A 0.000,B 0.000,C 90.000,E1 98.106} C_DIS
LIN {X 0.019,Y -477.732,Z 642.542,A 0.000,B 0.000,C 90.000,E1 97.587} C_DIS
LIN {X 0.169,Y -476.538,Z 642.539,A 0.000,B 0.000,C 90.000,E1 97.068} C_DIS
LIN {X 0.036,Y -475.510,Z 642.538,A 0.000,B 0.000,C 90.000,E1 96.834} C_DIS
LIN {X -0.154,Y -474.128,Z 642.537,A 0.000,B 0.000,C 90.000,E1 96.606} C_DIS
LIN {X -0.143,Y -456.868,Z 642.523,A 0.000,B 0.000,C 90.000,E1 94.069} C_DIS
LIN {X 0.035,Y -446.071,Z 642.512,A 0.000,B 0.000,C 90.000,E1 92.236} C_DIS
LIN {X 0.168,Y -434.582,Z 642.501,A 0.000,B 0.000,C 90.000,E1 90.115} C_DIS
LIN {X 0.057,Y -427.164,Z 642.493,A 0.000,B 0.000,C 90.000,E1 88.797} C_DIS
LIN {X -0.041,Y -417.867,Z 642.484,A 0.000,B 0.000,C 90.000,E1 87.192} C_DIS
LIN {X -0.102,Y -405.397,Z 642.472,A 0.000,B 0.000,C 90.000,E1 85.008} C_DIS
LIN {X 0.057,Y -390.216,Z 642.457,A 0.000,B 0.000,C 90.000,E1 82.186} C_DIS
END
